LIN {X 0,Y 524.085,Z 47.2,A -85,B 0,C 180,E1 -4854.614,E2 -4854.614} C_VEL
LIN {X 0,Y 524.114,Z 47.199,A -85,B 0,C 180,E1 -4857.694,E2 -4857.694} C_VEL
LIN {X 0,Y 524.126,Z 47.193,A -85,B 0,C 180,E1 -4860.768,E2 -4860.768} C_VEL
LIN {X 0,Y 524.073,Z 47.2,A -85,B 0,C 180,E1 -4863.075,E2 -4863.075} C_VEL
LIN {X 0,Y 524.02,Z 47.208,A -85,B 0,C 180,E1 -4866.159,E2 -4866.159} C_VEL
LIN {X 0,Y 523.989,Z 47.214,A -85,B 0,C 180,E1 -4869.262,E2 -4869.262} C_VEL
LIN {X 0,Y 524.007,Z 47.211,A -85,B 0,C 180,E1 -4871.739,E2 -4871.739} C_VEL
LIN {X 0,Y 523.998,Z 47.213,A -85,B 0,C 180,E1 -4875.052,E2 -4875.052} C_VEL
LIN {X 0,Y 523.949,Z 47.214,A -85,B 0,C 180,E1 -4877.969,E2 -4877.969} C_VEL
LIN {X 0,Y 523.976,Z 47.213,A -85,B 0,C 180,E1 -4880.41,E2 -4880.41} C_VEL
LIN {X 0,Y 523.914,Z 47.225,A -85,B 0,C 180,E1 -4882.893,E2 -4882.893} C_VEL
LIN {X 0,Y 523.938,Z 47.218,A -85,B 0,C 180,E1 -4885.419,E2 -4885.419} C_VEL
LIN {X 0,Y 523.921,Z 47.219,A -85,B 0,C 180,E1 -4888.002,E2 -4888.002} C_VEL
LIN {X 0,Y 523.948,Z 47.22,A -85,B 0,C 180,E1 -4890.854,E2 -4890.854} C_VEL
LIN {X 0,Y 523.932,Z 47.218,A -85,B 0,C 180,E1 -4893.729,E2 -4893.729} C_VEL
LIN {X 0,Y 523.9,Z 47.228,A -85,B 0,C 180,E1 -4896.4,E2 -4896.4} C_VEL
LIN {X 0,Y 523.921,Z 47.219,A -85,B 0,C 180,E1 -4899.085,E2 -4899.085} C_VEL
LIN {X 0,Y 523.942,Z 47.222,A -85,B 0,C 180,E1 -4902.12,E2 -4902.12} C_VEL
LIN {X 0,Y 523.94,Z 47.218,A -85,B 0,C 180,E1 -4905.311,E2 -4905.311} C_VEL
LIN {X 0,Y 523.893,Z 47.223,A -85,B 0,C 180,E1 -4906.9,E2 -4906.9} C_VEL
LIN {X 0,Y 523.23,Z 47.311,A -85,B 0,C 180,E1 -4907.542,E2 -4907.542} C_VEL
LIN {X 0,Y 520.385,Z 47.666,A -85,B 0,C 180,E1 -4908.583,E2 -4908.583} C_VEL
LIN {X 0,Y 517.978,Z 47.966,A -85,B 0,C 180,E1 -4909.423,E2 -4909.423} C_VEL
LIN {X 0,Y 516.946,Z 48.093,A -85,B 0,C 180,E1 -4910.07,E2 -4910.07} C_VEL
LIN {X 0,Y 516.863,Z 48.101,A -85,B 0,C 180,E1 -4910.29,E2 -4910.29} C_VEL
LIN {X 0,Y 516.854,Z 48.105,A -85,B 0,C 180,E1 -4913.347,E2 -4913.347} C_VEL
LIN {X 0,Y 516.885,Z 48.1,A -85,B 0,C 180,E1 -4916.119,E2 -4916.119} C_VEL
LIN {X 0,Y 516.89,Z 48.102,A -85,B 0,C 180,E1 -4918.936,E2 -4918.936} C_VEL
LIN {X 0,Y 516.943,Z 48.197,A -85,B 0,C 180,E1 -4921.475,E2 -4921.475} C_VEL
LIN {X 0,Y 517.512,Z 52.987,A -85,B 0,C 180,E1 -4922.501,E2 -4922.501} C_VEL
LIN {X 0,Y 517.34,Z 63.587,A -85,B 0,C 180,E1 -4924.686,E2 -4924.686} C_VEL
LIN {X 0,Y 519.23,Z 73.369,A -85,B 0,C 180,E1 -4924.897,E2 -4924.897} C_VEL
LIN {X 0,Y 518.679,Z 169.72,A -85,B 0,C 180,E1 -4926.254,E2 -4926.254} C_VEL
LIN {X 0,Y 518.545,Z 182.73,A -85,B 0,C 180,E1 -4926.592,E2 -4926.592} C_VEL
LIN {X 0,Y 518.389,Z 194.491,A -85,B 0,C 180,E1 -4927.042,E2 -4927.042} C_VEL
LIN {X 0,Y 518.056,Z 206.81,A -85,B 0,C 180,E1 -4927.675,E2 -4927.675} C_VEL
LIN {X 0,Y 517.756,Z 217.555,A -85,B 0,C 180,E1 -4928.396,E2 -4928.396} C_VEL
LIN {X 0,Y 517.473,Z 228.558,A -85,B 0,C 180,E1 -4929.322,E2 -4929.322} C_VEL
LIN {X 0,Y 517.175,Z 238.359,A -85,B 0,C 180,E1 -4930.346,E2 -4930.346} C_VEL
LIN {X 0,Y 516.894,Z 247.673,A -85,B 0,C 180,E1 -4931.571,E2 -4931.571} C_VEL
LIN {X 0,Y 516.723,Z 255.105,A -85,B 0,C 180,E1 -4932.793,E2 -4932.793} C_VEL
LIN {X 0,Y 516.573,Z 260.062,A -85,B 0,C 180,E1 -4933.805,E2 -4933.805} C_VEL
LIN {X 0,Y 516.466,Z 264.958,A -85,B 0,C 180,E1 -4935.052,E2 -4935.052} C_VEL
LIN {X 0,Y 516.358,Z 268.425,A -85,B 0,C 180,E1 -4936.22,E2 -4936.22} C_VEL
LIN {X 0,Y 516.301,Z 270.961,A -85,B 0,C 180,E1 -4937.42,E2 -4937.42} C_VEL
LIN {X 0,Y 516.284,Z 272.456,A -85,B 0,C 180,E1 -4938.554,E2 -4938.554} C_VEL
LIN {X 0,Y 516.265,Z 273.148,A -85,B 0,C 180,E1 -4939.807,E2 -4939.807} C_VEL
LIN {X 0,Y 516.232,Z 273.083,A -85,B 0,C 180,E1 -4940.598,E2 -4940.598} C_VEL
LIN {X 0,Y 516.285,Z 272.595,A -85,B 0,C 180,E1 -4941.388,E2 -4941.388} C_VEL
LIN {X 0,Y 516.367,Z 270.394,A -85,B 0,C 180,E1 -4942.964,E2 -4942.964} C_VEL
LIN {X 0,Y 516.433,Z 267.658,A -85,B 0,C 180,E1 -4944.142,E2 -4944.142} C_VEL
LIN {X 0,Y 516.477,Z 263.923,A -85,B 0,C 180,E1 -4945.317,E2 -4945.317} C_VEL
LIN {X 0,Y 516.581,Z 259.084,A -85,B 0,C 180,E1 -4946.49,E2 -4946.49} C_VEL
LIN {X 0,Y 516.689,Z 253.013,A -85,B 0,C 180,E1 -4947.661,E2 -4947.661} C_VEL
LIN {X 0,Y 516.952,Z 245.461,A -85,B 0,C 180,E1 -4948.832,E2 -4948.832} C_VEL
LIN {X 0,Y 517.195,Z 236.016,A -85,B 0,C 180,E1 -4950,E2 -4950} C_VEL
LIN {X 0,Y 517.501,Z 226.287,A -85,B 0,C 180,E1 -4950.973,E2 -4950.973} C_VEL
LIN {X 0,Y 517.809,Z 215.383,A -85,B 0,C 180,E1 -4951.847,E2 -4951.847} C_VEL
LIN {X 0,Y 518.15,Z 204.714,A -85,B 0,C 180,E1 -4952.527,E2 -4952.527} C_VEL
LIN {X 0,Y 518.365,Z 193.027,A -85,B 0,C 180,E1 -4953.109,E2 -4953.109} C_VEL
LIN {X 0,Y 518.526,Z 180.438,A -85,B 0,C 180,E1 -4953.57,E2 -4953.57} C_VEL
LIN {X 0,Y 518.713,Z 168.16,A -85,B 0,C 180,E1 -4953.86,E2 -4953.86} C_VEL
LIN {X 0,Y 519.005,Z 71.995,A -85,B 0,C 180,E1 -4955.214,E2 -4955.214} C_VEL
LIN {X 0,Y 517.288,Z 63.413,A -85,B 0,C 180,E1 -4955.409,E2 -4955.409} C_VEL
LIN {X 0,Y 517.555,Z 52.863,A -85,B 0,C 180,E1 -4957.57,E2 -4957.57} C_VEL
LIN {X 0,Y 516.967,Z 48.094,A -85,B 0,C 180,E1 -4958.6,E2 -4958.6} C_VEL
LIN {X 0,Y 516.954,Z 48.086,A -85,B 0,C 180,E1 -4961.807,E2 -4961.807} C_VEL
LIN {X 0,Y 516.949,Z 48.088,A -85,B 0,C 180,E1 -4965.148,E2 -4965.148} C_VEL
LIN {X 0,Y 516.927,Z 48.095,A -85,B 0,C 180,E1 -4968.222,E2 -4968.222} C_VEL
LIN {X 0,Y 516.914,Z 48.095,A -85,B 0,C 180,E1 -4970.702,E2 -4970.702} C_VEL
LIN {X 0,Y 516.893,Z 48.1,A -85,B 0,C 180,E1 -4974.073,E2 -4974.073} C_VEL
LIN {X 0,Y 516.928,Z 48.091,A -85,B 0,C 180,E1 -4976.658,E2 -4976.658} C_VEL
LIN {X 0,Y 516.913,Z 48.093,A -85,B 0,C 180,E1 -4979.524,E2 -4979.524} C_VEL
LIN {X 0,Y 516.898,Z 48.094,A -85,B 0,C 180,E1 -4982.544,E2 -4982.544} C_VEL
LIN {X 0,Y 516.882,Z 48.097,A -85,B 0,C 180,E1 -4985.332,E2 -4985.332} C_VEL
LIN {X 0,Y 516.883,Z 48.101,A -85,B 0,C 180,E1 -4987.943,E2 -4987.943} C_VEL
LIN {X 0,Y 516.886,Z 48.095,A -85,B 0,C 180,E1 -4990.742,E2 -4990.742} C_VEL
LIN {X 0,Y 516.885,Z 48.095,A -85,B 0,C 180,E1 -4992.832,E2 -4992.832} C_VEL
LIN {X 0,Y 516.898,Z 48.096,A -85,B 0,C 180,E1 -4995.007,E2 -4995.007} C_VEL
LIN {X 0,Y 516.916,Z 48.091,A -85,B 0,C 180,E1 -4998.399,E2 -4998.399} C_VEL
LIN {X 0,Y 516.884,Z 48.103,A -85,B 0,C 180,E1 -5001.284,E2 -5001.284} C_VEL
LIN {X 0,Y 516.876,Z 48.096,A -85,B 0,C 180,E1 -5004.22,E2 -5004.22} C_VEL
LIN {X 0,Y 516.899,Z 48.102,A -85,B 0,C 180,E1 -5007.053,E2 -5007.053} C_VEL
LIN {X 0,Y 516.896,Z 48.093,A -85,B 0,C 180,E1 -5009.797,E2 -5009.797} C_VEL
LIN {X 0,Y 516.931,Z 48.093,A -85,B 0,C 180,E1 -5012.468,E2 -5012.468} C_VEL
LIN {X 0,Y 516.908,Z 48.096,A -85,B 0,C 180,E1 -5015.072,E2 -5015.072} C_VEL
LIN {X 0,Y 516.891,Z 48.1,A -85,B 0,C 180,E1 -5018.463,E2 -5018.463} C_VEL
LIN {X 0,Y 516.899,Z 48.096,A -85,B 0,C 180,E1 -5020.955,E2 -5020.955} C_VEL
LIN {X 0,Y 516.907,Z 48.092,A -85,B 0,C 180,E1 -5023.41,E2 -5023.41} C_VEL
LIN {X 0,Y 516.9,Z 48.095,A -85,B 0,C 180,E1 -5025.834,E2 -5025.834} C_VEL
LIN {X 0,Y 516.972,Z 48.092,A -85,B 0,C 180,E1 -5028.234,E2 -5028.234} C_VEL
LIN {X 0,Y 516.961,Z 48.086,A -85,B 0,C 180,E1 -5031.4,E2 -5031.4} C_VEL
LIN {X 0,Y 517.015,Z 48.083,A -85,B 0,C 180,E1 -5033.757,E2 -5033.757} C_VEL
LIN {X 0,Y 517.086,Z 48.074,A -85,B 0,C 180,E1 -5037.663,E2 -5037.663} C_VEL
LIN {X 0,Y 517.098,Z 48.068,A -85,B 0,C 180,E1 -5040.779,E2 -5040.779} C_VEL
LIN {X 0,Y 517.015,Z 48.08,A -85,B 0,C 180,E1 -5043.117,E2 -5043.117} C_VEL
LIN {X 0,Y 516.982,Z 48.084,A -85,B 0,C 180,E1 -5046.244,E2 -5046.244} C_VEL
LIN {X 0,Y 516.947,Z 48.094,A -85,B 0,C 180,E1 -5049.389,E2 -5049.389} C_VEL
LIN {X 0,Y 516.958,Z 48.089,A -85,B 0,C 180,E1 -5051.807,E2 -5051.807} C_VEL
LIN {X 0,Y 516.951,Z 48.093,A -85,B 0,C 180,E1 -5055.146,E2 -5055.146} C_VEL
LIN {X 0,Y 516.919,Z 48.09,A -85,B 0,C 180,E1 -5058.223,E2 -5058.223} C_VEL
LIN {X 0,Y 516.918,Z 48.094,A -85,B 0,C 180,E1 -5060.701,E2 -5060.701} C_VEL
LIN {X 0,Y 516.895,Z 48.093,A -85,B 0,C 180,E1 -5064.073,E2 -5064.073} C_VEL
LIN {X 0,Y 516.904,Z 48.098,A -85,B 0,C 180,E1 -5066.659,E2 -5066.659} C_VEL
LIN {X 0,Y 516.916,Z 48.091,A -85,B 0,C 180,E1 -5069.524,E2 -5069.524} C_VEL
LIN {X 0,Y 516.899,Z 48.1,A -85,B 0,C 180,E1 -5072.543,E2 -5072.543} C_VEL
LIN {X 0,Y 516.868,Z 48.097,A -85,B 0,C 180,E1 -5075.329,E2 -5075.329} C_VEL
LIN {X 0,Y 516.883,Z 48.097,A -85,B 0,C 180,E1 -5077.943,E2 -5077.943} C_VEL
LIN {X 0,Y 516.887,Z 48.098,A -85,B 0,C 180,E1 -5080.742,E2 -5080.742} C_VEL
LIN {X 0,Y 516.886,Z 48.097,A -85,B 0,C 180,E1 -5082.831,E2 -5082.831} C_VEL
LIN {X 0,Y 516.899,Z 48.093,A -85,B 0,C 180,E1 -5085.007,E2 -5085.007} C_VEL
LIN {X 0,Y 516.913,Z 48.096,A -85,B 0,C 180,E1 -5088.399,E2 -5088.399} C_VEL
LIN {X 0,Y 516.881,Z 48.096,A -85,B 0,C 180,E1 -5091.284,E2 -5091.284} C_VEL
LIN {X 0,Y 516.872,Z 48.101,A -85,B 0,C 180,E1 -5094.219,E2 -5094.219} C_VEL
LIN {X 0,Y 516.885,Z 48.095,A -85,B 0,C 180,E1 -5097.052,E2 -5097.052} C_VEL
LIN {X 0,Y 516.891,Z 48.103,A -85,B 0,C 180,E1 -5099.796,E2 -5099.796} C_VEL
LIN {X 0,Y 516.928,Z 48.092,A -85,B 0,C 180,E1 -5102.467,E2 -5102.467} C_VEL
LIN {X 0,Y 516.956,Z 48.23,A -85,B 0,C 180,E1 -5104.563,E2 -5104.563} C_VEL
LIN {X 0,Y 518.456,Z 56.174,A -85,B 0,C 180,E1 -5105.835,E2 -5105.835} C_VEL
LIN {X 0,Y 518.141,Z 71.265,A -85,B 0,C 180,E1 -5108.099,E2 -5108.099} C_VEL
LIN {X 0,Y 517.746,Z 90.754,A -85,B 0,C 180,E1 -5110.987,E2 -5110.987} C_VEL
LIN {X 0,Y 517.313,Z 110.152,A -85,B 0,C 180,E1 -5113.829,E2 -5113.829} C_VEL
LIN {X 0,Y 517.228,Z 115.912,A -85,B 0,C 180,E1 -5114.631,E2 -5114.631} C_VEL
LIN {X 0,Y 519.045,Z 128.632,A -85,B 0,C 180,E1 -5114.862,E2 -5114.862} C_VEL
LIN {X 0,Y 518.57,Z 224.217,A -85,B 0,C 180,E1 -5116.205,E2 -5116.205} C_VEL
LIN {X 0,Y 518.303,Z 237.571,A -85,B 0,C 180,E1 -5116.548,E2 -5116.548} C_VEL
LIN {X 0,Y 518.026,Z 250.921,A -85,B 0,C 180,E1 -5117.064,E2 -5117.064} C_VEL
LIN {X 0,Y 517.698,Z 262.803,A -85,B 0,C 180,E1 -5117.696,E2 -5117.696} C_VEL
LIN {X 0,Y 517.432,Z 273.773,A -85,B 0,C 180,E1 -5118.443,E2 -5118.443} C_VEL
LIN {X 0,Y 517.159,Z 284.265,A -85,B 0,C 180,E1 -5119.329,E2 -5119.329} C_VEL
LIN {X 0,Y 516.841,Z 292.841,A -85,B 0,C 180,E1 -5120.213,E2 -5120.213} C_VEL
LIN {X 0,Y 516.653,Z 300.762,A -85,B 0,C 180,E1 -5121.197,E2 -5121.197} C_VEL
LIN {X 0,Y 516.502,Z 308.503,A -85,B 0,C 180,E1 -5122.376,E2 -5122.376} C_VEL
LIN {X 0,Y 516.353,Z 315.637,A -85,B 0,C 180,E1 -5123.749,E2 -5123.749} C_VEL
LIN {X 0,Y 516.311,Z 320.386,A -85,B 0,C 180,E1 -5124.924,E2 -5124.924} C_VEL
LIN {X 0,Y 516.369,Z 324.019,A -85,B 0,C 180,E1 -5126.098,E2 -5126.098} C_VEL
LIN {X 0,Y 516.327,Z 325.889,A -85,B 0,C 180,E1 -5126.879,E2 -5126.879} C_VEL
LIN {X 0,Y 516.266,Z 327.289,A -85,B 0,C 180,E1 -5127.659,E2 -5127.659} C_VEL
LIN {X 0,Y 516.189,Z 328.895,A -85,B 0,C 180,E1 -5129.22,E2 -5129.22} C_VEL
LIN {X 0,Y 516.194,Z 329.111,A -85,B 0,C 180,E1 -5130,E2 -5130} C_VEL
LIN {X 0,Y 516.189,Z 328.892,A -85,B 0,C 180,E1 -5130.78,E2 -5130.78} C_VEL
LIN {X 0,Y 516.266,Z 327.279,A -85,B 0,C 180,E1 -5132.341,E2 -5132.341} C_VEL
LIN {X 0,Y 516.327,Z 325.875,A -85,B 0,C 180,E1 -5133.121,E2 -5133.121} C_VEL
LIN {X 0,Y 516.311,Z 322.917,A -85,B 0,C 180,E1 -5134.293,E2 -5134.293} C_VEL
LIN {X 0,Y 516.363,Z 318.916,A -85,B 0,C 180,E1 -5135.467,E2 -5135.467} C_VEL
LIN {X 0,Y 516.406,Z 313.117,A -85,B 0,C 180,E1 -5136.771,E2 -5136.771} C_VEL
LIN {X 0,Y 516.558,Z 306.047,A -85,B 0,C 180,E1 -5138.016,E2 -5138.016} C_VEL
LIN {X 0,Y 516.724,Z 297.714,A -85,B 0,C 180,E1 -5139.196,E2 -5139.196} C_VEL
LIN {X 0,Y 516.941,Z 289.178,A -85,B 0,C 180,E1 -5140.18,E2 -5140.18} C_VEL
LIN {X 0,Y 517.291,Z 278.64,A -85,B 0,C 180,E1 -5141.163,E2 -5141.163} C_VEL
LIN {X 0,Y 517.566,Z 267.025,A -85,B 0,C 180,E1 -5142.034,E2 -5142.034} C_VEL
LIN {X 0,Y 517.903,Z 254.859,A -85,B 0,C 180,E1 -5142.739,E2 -5142.739} C_VEL
LIN {X 0,Y 518.195,Z 242.464,A -85,B 0,C 180,E1 -5143.28,E2 -5143.28} C_VEL
LIN {X 0,Y 518.456,Z 229.739,A -85,B 0,C 180,E1 -5143.673,E2 -5143.673} C_VEL
LIN {X 0,Y 518.648,Z 214.605,A -85,B 0,C 180,E1 -5143.942,E2 -5143.942} C_VEL
LIN {X 0,Y 518.957,Z 128.068,A -85,B 0,C 180,E1 -5145.147,E2 -5145.147} C_VEL
LIN {X 0,Y 517.216,Z 115.441,A -85,B 0,C 180,E1 -5145.386,E2 -5145.386} C_VEL
LIN {X 0,Y 517.714,Z 93.474,A -85,B 0,C 180,E1 -5148.603,E2 -5148.603} C_VEL
LIN {X 0,Y 518.102,Z 74.124,A -85,B 0,C 180,E1 -5151.485,E2 -5151.485} C_VEL
LIN {X 0,Y 518.546,Z 56.468,A -85,B 0,C 180,E1 -5154.16,E2 -5154.16} C_VEL
LIN {X 0,Y 516.956,Z 48.092,A -85,B 0,C 180,E1 -5155.572,E2 -5155.572} C_VEL
LIN {X 0,Y 516.919,Z 48.098,A -85,B 0,C 180,E1 -5158.415,E2 -5158.415} C_VEL
LIN {X 0,Y 516.892,Z 48.095,A -85,B 0,C 180,E1 -5161.11,E2 -5161.11} C_VEL
LIN {X 0,Y 516.89,Z 48.102,A -85,B 0,C 180,E1 -5163.963,E2 -5163.963} C_VEL
LIN {X 0,Y 516.88,Z 48.097,A -85,B 0,C 180,E1 -5166.746,E2 -5166.746} C_VEL
LIN {X 0,Y 516.885,Z 48.098,A -85,B 0,C 180,E1 -5169.721,E2 -5169.721} C_VEL
LIN {X 0,Y 516.915,Z 48.099,A -85,B 0,C 180,E1 -5171.775,E2 -5171.775} C_VEL
LIN {X 0,Y 516.898,Z 48.093,A -85,B 0,C 180,E1 -5175.007,E2 -5175.007} C_VEL
LIN {X 0,Y 516.917,Z 48.09,A -85,B 0,C 180,E1 -5178.399,E2 -5178.399} C_VEL
LIN {X 0,Y 516.884,Z 48.1,A -85,B 0,C 180,E1 -5181.284,E2 -5181.284} C_VEL
LIN {X 0,Y 516.875,Z 48.096,A -85,B 0,C 180,E1 -5184.22,E2 -5184.22} C_VEL
LIN {X 0,Y 516.885,Z 48.1,A -85,B 0,C 180,E1 -5187.052,E2 -5187.052} C_VEL
LIN {X 0,Y 516.896,Z 48.092,A -85,B 0,C 180,E1 -5189.796,E2 -5189.796} C_VEL
LIN {X 0,Y 516.931,Z 48.092,A -85,B 0,C 180,E1 -5192.467,E2 -5192.467} C_VEL
LIN {X 0,Y 516.908,Z 48.098,A -85,B 0,C 180,E1 -5195.072,E2 -5195.072} C_VEL
LIN {X 0,Y 516.89,Z 48.098,A -85,B 0,C 180,E1 -5198.462,E2 -5198.462} C_VEL
LIN {X 0,Y 516.899,Z 48.097,A -85,B 0,C 180,E1 -5200.955,E2 -5200.955} C_VEL
LIN {X 0,Y 516.915,Z 48.089,A -85,B 0,C 180,E1 -5203.41,E2 -5203.41} C_VEL
LIN {X 0,Y 516.899,Z 48.095,A -85,B 0,C 180,E1 -5205.834,E2 -5205.834} C_VEL
LIN {X 0,Y 516.971,Z 48.089,A -85,B 0,C 180,E1 -5208.234,E2 -5208.234} C_VEL
LIN {X 0,Y 516.97,Z 48.085,A -85,B 0,C 180,E1 -5211.4,E2 -5211.4} C_VEL
LIN {X 0,Y 517.014,Z 48.079,A -85,B 0,C 180,E1 -5213.757,E2 -5213.757} C_VEL
LIN {X 0,Y 517.085,Z 48.074,A -85,B 0,C 180,E1 -5217.663,E2 -5217.663} C_VEL
LIN {X 0,Y 517.097,Z 48.069,A -85,B 0,C 180,E1 -5220.779,E2 -5220.779} C_VEL
LIN {X 0,Y 517.014,Z 48.079,A -85,B 0,C 180,E1 -5223.117,E2 -5223.117} C_VEL
LIN {X 0,Y 516.989,Z 48.083,A -85,B 0,C 180,E1 -5226.243,E2 -5226.243} C_VEL
LIN {X 0,Y 516.945,Z 48.092,A -85,B 0,C 180,E1 -5229.389,E2 -5229.389} C_VEL
LIN {X 0,Y 516.957,Z 48.089,A -85,B 0,C 180,E1 -5231.807,E2 -5231.807} C_VEL
LIN {X 0,Y 516.949,Z 48.092,A -85,B 0,C 180,E1 -5235.146,E2 -5235.146} C_VEL
LIN {X 0,Y 516.917,Z 48.09,A -85,B 0,C 180,E1 -5238.222,E2 -5238.222} C_VEL
LIN {X 0,Y 516.916,Z 48.096,A -85,B 0,C 180,E1 -5240.701,E2 -5240.701} C_VEL
LIN {X 0,Y 516.906,Z 48.092,A -85,B 0,C 180,E1 -5244.072,E2 -5244.072} C_VEL
LIN {X 0,Y 516.901,Z 48.1,A -85,B 0,C 180,E1 -5246.659,E2 -5246.659} C_VEL
LIN {X 0,Y 516.913,Z 48.092,A -85,B 0,C 180,E1 -5249.523,E2 -5249.523} C_VEL
LIN {X 0,Y 516.897,Z 48.101,A -85,B 0,C 180,E1 -5252.543,E2 -5252.543} C_VEL
LIN {X 0,Y 516.864,Z 48.098,A -85,B 0,C 180,E1 -5255.329,E2 -5255.329} C_VEL
LIN {X 0,Y 516.881,Z 48.099,A -85,B 0,C 180,E1 -5257.943,E2 -5257.943} C_VEL
LIN {X 0,Y 516.873,Z 48.094,A -85,B 0,C 180,E1 -5260.743,E2 -5260.743} C_VEL
LIN {X 0,Y 516.883,Z 48.103,A -85,B 0,C 180,E1 -5263.893,E2 -5263.893} C_VEL
LIN {X 0,Y 516.846,Z 48.101,A -85,B 0,C 180,E1 -5266.901,E2 -5266.901} C_VEL
LIN {X 0,Y 516.886,Z 48.102,A -85,B 0,C 180,E1 -5269.59,E2 -5269.59} C_VEL
LIN {X 0,Y 516.863,Z 48.101,A -85,B 0,C 180,E1 -5270.29,E2 -5270.29} C_VEL
LIN {X 0,Y 516.199,Z 48.182,A -85,B 0,C 180,E1 -5270.94,E2 -5270.94} C_VEL
LIN {X 0,Y 513.349,Z 48.543,A -85,B 0,C 180,E1 -5271.996,E2 -5271.996} C_VEL
LIN {X 0,Y 510.936,Z 48.848,A -85,B 0,C 180,E1 -5272.846,E2 -5272.846} C_VEL
LIN {X 0,Y 509.894,Z 48.976,A -85,B 0,C 180,E1 -5273.503,E2 -5273.503} C_VEL
LIN {X 0,Y 509.807,Z 48.984,A -85,B 0,C 180,E1 -5273.725,E2 -5273.725} C_VEL
LIN {X 0,Y 509.843,Z 48.976,A -85,B 0,C 180,E1 -5276.538,E2 -5276.538} C_VEL
LIN {X 0,Y 509.841,Z 48.982,A -85,B 0,C 180,E1 -5279.334,E2 -5279.334} C_VEL
LIN {X 0,Y 509.924,Z 49.163,A -85,B 0,C 180,E1 -5281.344,E2 -5281.344} C_VEL
LIN {X 0,Y 510.522,Z 54.689,A -85,B 0,C 180,E1 -5282.537,E2 -5282.537} C_VEL
LIN {X 0,Y 510.374,Z 63.959,A -85,B 0,C 180,E1 -5284.464,E2 -5284.464} C_VEL
LIN {X 0,Y 512.396,Z 74.105,A -85,B 0,C 180,E1 -5284.688,E2 -5284.688} C_VEL
LIN {X 0,Y 511.831,Z 169.609,A -85,B 0,C 180,E1 -5286.051,E2 -5286.051} C_VEL
LIN {X 0,Y 511.668,Z 182.796,A -85,B 0,C 180,E1 -5286.392,E2 -5286.392} C_VEL
LIN {X 0,Y 511.491,Z 194.615,A -85,B 0,C 180,E1 -5286.848,E2 -5286.848} C_VEL
LIN {X 0,Y 511.164,Z 206.558,A -85,B 0,C 180,E1 -5287.465,E2 -5287.465} C_VEL
LIN {X 0,Y 510.842,Z 217.454,A -85,B 0,C 180,E1 -5288.194,E2 -5288.194} C_VEL
LIN {X 0,Y 510.543,Z 227.421,A -85,B 0,C 180,E1 -5289.028,E2 -5289.028} C_VEL
LIN {X 0,Y 510.239,Z 237.494,A -85,B 0,C 180,E1 -5290.068,E2 -5290.068} C_VEL
LIN {X 0,Y 509.956,Z 245.666,A -85,B 0,C 180,E1 -5291.103,E2 -5291.103} C_VEL
LIN {X 0,Y 509.706,Z 253.551,A -85,B 0,C 180,E1 -5292.341,E2 -5292.341} C_VEL
LIN {X 0,Y 509.531,Z 259.805,A -85,B 0,C 180,E1 -5293.575,E2 -5293.575} C_VEL
LIN {X 0,Y 509.384,Z 265.306,A -85,B 0,C 180,E1 -5294.971,E2 -5294.971} C_VEL
LIN {X 0,Y 509.321,Z 268.434,A -85,B 0,C 180,E1 -5296.026,E2 -5296.026} C_VEL
LIN {X 0,Y 509.214,Z 271.091,A -85,B 0,C 180,E1 -5297.242,E2 -5297.242} C_VEL
LIN {X 0,Y 509.211,Z 272.807,A -85,B 0,C 180,E1 -5298.5,E2 -5298.5} C_VEL
LIN {X 0,Y 509.197,Z 273.504,A -85,B 0,C 180,E1 -5299.664,E2 -5299.664} C_VEL
LIN {X 0,Y 509.183,Z 273.096,A -85,B 0,C 180,E1 -5301.267,E2 -5301.267} C_VEL
LIN {X 0,Y 509.231,Z 272.268,A -85,B 0,C 180,E1 -5302.067,E2 -5302.067} C_VEL
LIN {X 0,Y 509.318,Z 269.817,A -85,B 0,C 180,E1 -5303.473,E2 -5303.473} C_VEL
LIN {X 0,Y 509.327,Z 266.123,A -85,B 0,C 180,E1 -5304.854,E2 -5304.854} C_VEL
LIN {X 0,Y 509.501,Z 261.783,A -85,B 0,C 180,E1 -5306.045,E2 -5306.045} C_VEL
LIN {X 0,Y 509.555,Z 256.296,A -85,B 0,C 180,E1 -5307.233,E2 -5307.233} C_VEL
LIN {X 0,Y 509.829,Z 249.438,A -85,B 0,C 180,E1 -5308.42,E2 -5308.42} C_VEL
LIN {X 0,Y 510.083,Z 240.879,A -85,B 0,C 180,E1 -5309.605,E2 -5309.605} C_VEL
LIN {X 0,Y 510.324,Z 232.146,A -85,B 0,C 180,E1 -5310.592,E2 -5310.592} C_VEL
LIN {X 0,Y 510.708,Z 221.386,A -85,B 0,C 180,E1 -5311.577,E2 -5311.577} C_VEL
LIN {X 0,Y 511.043,Z 210.526,A -85,B 0,C 180,E1 -5312.365,E2 -5312.365} C_VEL
LIN {X 0,Y 511.349,Z 198.405,A -85,B 0,C 180,E1 -5313.053,E2 -5313.053} C_VEL
LIN {X 0,Y 511.588,Z 185.604,A -85,B 0,C 180,E1 -5313.594,E2 -5313.594} C_VEL
LIN {X 0,Y 511.751,Z 172.634,A -85,B 0,C 180,E1 -5313.962,E2 -5313.962} C_VEL
LIN {X 0,Y 511.935,Z 152.544,A -85,B 0,C 180,E1 -5314.281,E2 -5314.281} C_VEL
LIN {X 0,Y 512.204,Z 73.139,A -85,B 0,C 180,E1 -5315.404,E2 -5315.404} C_VEL
LIN {X 0,Y 510.315,Z 63.795,A -85,B 0,C 180,E1 -5315.607,E2 -5315.607} C_VEL
LIN {X 0,Y 510.561,Z 53.878,A -85,B 0,C 180,E1 -5317.651,E2 -5317.651} C_VEL
LIN {X 0,Y 509.913,Z 48.973,A -85,B 0,C 180,E1 -5318.72,E2 -5318.72} C_VEL
LIN {X 0,Y 509.906,Z 48.964,A -85,B 0,C 180,E1 -5321.932,E2 -5321.932} C_VEL
LIN {X 0,Y 509.896,Z 48.966,A -85,B 0,C 180,E1 -5325.242,E2 -5325.242} C_VEL
LIN {X 0,Y 509.884,Z 48.97,A -85,B 0,C 180,E1 -5327.999,E2 -5327.999} C_VEL
LIN {X 0,Y 509.852,Z 48.972,A -85,B 0,C 180,E1 -5331.002,E2 -5331.002} C_VEL
LIN {X 0,Y 509.824,Z 48.975,A -85,B 0,C 180,E1 -5333.564,E2 -5333.564} C_VEL
LIN {X 0,Y 509.914,Z 48.968,A -85,B 0,C 180,E1 -5336.379,E2 -5336.379} C_VEL
LIN {X 0,Y 509.879,Z 48.968,A -85,B 0,C 180,E1 -5338.844,E2 -5338.844} C_VEL
LIN {X 0,Y 509.823,Z 48.978,A -85,B 0,C 180,E1 -5341.59,E2 -5341.59} C_VEL
LIN {X 0,Y 509.855,Z 48.972,A -85,B 0,C 180,E1 -5344.414,E2 -5344.414} C_VEL
LIN {X 0,Y 509.821,Z 48.978,A -85,B 0,C 180,E1 -5347.341,E2 -5347.341} C_VEL
LIN {X 0,Y 509.841,Z 48.973,A -85,B 0,C 180,E1 -5350.382,E2 -5350.382} C_VEL
LIN {X 0,Y 509.825,Z 48.977,A -85,B 0,C 180,E1 -5353.062,E2 -5353.062} C_VEL
LIN {X 0,Y 509.825,Z 48.978,A -85,B 0,C 180,E1 -5355.794,E2 -5355.794} C_VEL
LIN {X 0,Y 509.858,Z 48.971,A -85,B 0,C 180,E1 -5358.575,E2 -5358.575} C_VEL
LIN {X 0,Y 509.854,Z 48.972,A -85,B 0,C 180,E1 -5361.787,E2 -5361.787} C_VEL
LIN {X 0,Y 509.836,Z 48.975,A -85,B 0,C 180,E1 -5364.622,E2 -5364.622} C_VEL
LIN {X 0,Y 509.865,Z 48.972,A -85,B 0,C 180,E1 -5367.481,E2 -5367.481} C_VEL
LIN {X 0,Y 509.863,Z 48.971,A -85,B 0,C 180,E1 -5370.274,E2 -5370.274} C_VEL
LIN {X 0,Y 509.888,Z 48.973,A -85,B 0,C 180,E1 -5372.945,E2 -5372.945} C_VEL
LIN {X 0,Y 509.86,Z 48.97,A -85,B 0,C 180,E1 -5375.574,E2 -5375.574} C_VEL
LIN {X 0,Y 509.855,Z 48.974,A -85,B 0,C 180,E1 -5378.999,E2 -5378.999} C_VEL
LIN {X 0,Y 509.863,Z 48.969,A -85,B 0,C 180,E1 -5381.516,E2 -5381.516} C_VEL
LIN {X 0,Y 509.916,Z 48.966,A -85,B 0,C 180,E1 -5384.819,E2 -5384.819} C_VEL
LIN {X 0,Y 509.907,Z 48.97,A -85,B 0,C 180,E1 -5388.124,E2 -5388.124} C_VEL
LIN {X 0,Y 509.909,Z 48.964,A -85,B 0,C 180,E1 -5391.28,E2 -5391.28} C_VEL
LIN {X 0,Y 509.965,Z 48.96,A -85,B 0,C 180,E1 -5393.67,E2 -5393.67} C_VEL
LIN {X 0,Y 510.056,Z 48.95,A -85,B 0,C 180,E1 -5397.631,E2 -5397.631} C_VEL
LIN {X 0,Y 510.061,Z 48.951,A -85,B 0,C 180,E1 -5400,E2 -5400} C_VEL
LIN {X 0,Y 510.058,Z 48.947,A -85,B 0,C 180,E1 -5402.369,E2 -5402.369} C_VEL
LIN {X 0,Y 509.972,Z 48.963,A -85,B 0,C 180,E1 -5405.536,E2 -5405.536} C_VEL
LIN {X 0,Y 509.909,Z 48.964,A -85,B 0,C 180,E1 -5408.72,E2 -5408.72} C_VEL
LIN {X 0,Y 509.91,Z 48.966,A -85,B 0,C 180,E1 -5411.932,E2 -5411.932} C_VEL
LIN {X 0,Y 509.9,Z 48.973,A -85,B 0,C 180,E1 -5415.242,E2 -5415.242} C_VEL
LIN {X 0,Y 509.864,Z 48.97,A -85,B 0,C 180,E1 -5418.484,E2 -5418.484} C_VEL
LIN {X 0,Y 509.856,Z 48.978,A -85,B 0,C 180,E1 -5421.002,E2 -5421.002} C_VEL
LIN {X 0,Y 509.827,Z 48.976,A -85,B 0,C 180,E1 -5423.564,E2 -5423.564} C_VEL
LIN {X 0,Y 509.89,Z 48.968,A -85,B 0,C 180,E1 -5426.372,E2 -5426.372} C_VEL
LIN {X 0,Y 509.864,Z 48.969,A -85,B 0,C 180,E1 -5429.726,E2 -5429.726} C_VEL
LIN {X 0,Y 509.871,Z 48.976,A -85,B 0,C 180,E1 -5432.773,E2 -5432.773} C_VEL
LIN {X 0,Y 509.827,Z 48.974,A -85,B 0,C 180,E1 -5435.578,E2 -5435.578} C_VEL
LIN {X 0,Y 509.853,Z 48.977,A -85,B 0,C 180,E1 -5438.338,E2 -5438.338} C_VEL
LIN {X 0,Y 509.859,Z 48.97,A -85,B 0,C 180,E1 -5441.425,E2 -5441.425} C_VEL
LIN {X 0,Y 509.843,Z 48.975,A -85,B 0,C 180,E1 -5444.67,E2 -5444.67} C_VEL
LIN {X 0,Y 509.853,Z 48.979,A -85,B 0,C 180,E1 -5448.104,E2 -5448.104} C_VEL
LIN {X 0,Y 509.842,Z 48.973,A -85,B 0,C 180,E1 -5450.647,E2 -5450.647} C_VEL
LIN {X 0,Y 509.813,Z 48.98,A -85,B 0,C 180,E1 -5453.645,E2 -5453.645} C_VEL
LIN {X 0,Y 509.846,Z 48.972,A -85,B 0,C 180,E1 -5456.538,E2 -5456.538} C_VEL
LIN {X 0,Y 509.846,Z 48.975,A -85,B 0,C 180,E1 -5459.334,E2 -5459.334} C_VEL
LIN {X 0,Y 509.893,Z 48.971,A -85,B 0,C 180,E1 -5462.054,E2 -5462.054} C_VEL
LIN {X 0,Y 509.952,Z 49.138,A -85,B 0,C 180,E1 -5464.407,E2 -5464.407} C_VEL
LIN {X 0,Y 511.537,Z 58.216,A -85,B 0,C 180,E1 -5465.874,E2 -5465.874} C_VEL
LIN {X 0,Y 511.088,Z 76.393,A -85,B 0,C 180,E1 -5468.629,E2 -5468.629} C_VEL
LIN {X 0,Y 510.608,Z 98.096,A -85,B 0,C 180,E1 -5471.875,E2 -5471.875} C_VEL
LIN {X 0,Y 510.177,Z 115.209,A -85,B 0,C 180,E1 -5474.408,E2 -5474.408} C_VEL
LIN {X 0,Y 512.138,Z 129.834,A -85,B 0,C 180,E1 -5474.679,E2 -5474.679} C_VEL
LIN {X 0,Y 511.691,Z 223.748,A -85,B 0,C 180,E1 -5476.016,E2 -5476.016} C_VEL
LIN {X 0,Y 511.424,Z 236.376,A -85,B 0,C 180,E1 -5476.338,E2 -5476.338} C_VEL
LIN {X 0,Y 511.103,Z 249.378,A -85,B 0,C 180,E1 -5476.835,E2 -5476.835} C_VEL
LIN {X 0,Y 510.791,Z 261.177,A -85,B 0,C 180,E1 -5477.45,E2 -5477.45} C_VEL
LIN {X 0,Y 510.419,Z 272.08,A -85,B 0,C 180,E1 -5478.181,E2 -5478.181} C_VEL
LIN {X 0,Y 510.126,Z 282.798,A -85,B 0,C 180,E1 -5479.08,E2 -5479.08} C_VEL
LIN {X 0,Y 509.804,Z 292.454,A -85,B 0,C 180,E1 -5480.077,E2 -5480.077} C_VEL
LIN {X 0,Y 509.601,Z 300.377,A -85,B 0,C 180,E1 -5481.074,E2 -5481.074} C_VEL
LIN {X 0,Y 509.415,Z 308.117,A -85,B 0,C 180,E1 -5482.269,E2 -5482.269} C_VEL
LIN {X 0,Y 509.26,Z 315.252,A -85,B 0,C 180,E1 -5483.661,E2 -5483.661} C_VEL
LIN {X 0,Y 509.239,Z 320.003,A -85,B 0,C 180,E1 -5484.853,E2 -5484.853} C_VEL
LIN {X 0,Y 509.275,Z 323.635,A -85,B 0,C 180,E1 -5486.043,E2 -5486.043} C_VEL
LIN {X 0,Y 509.241,Z 325.506,A -85,B 0,C 180,E1 -5486.835,E2 -5486.835} C_VEL
LIN {X 0,Y 509.196,Z 326.907,A -85,B 0,C 180,E1 -5487.627,E2 -5487.627} C_VEL
LIN {X 0,Y 509.101,Z 328.512,A -85,B 0,C 180,E1 -5489.209,E2 -5489.209} C_VEL
LIN {X 0,Y 509.105,Z 328.727,A -85,B 0,C 180,E1 -5490,E2 -5490} C_VEL
LIN {X 0,Y 509.12,Z 327.895,A -85,B 0,C 180,E1 -5491.582,E2 -5491.582} C_VEL
LIN {X 0,Y 509.196,Z 326.894,A -85,B 0,C 180,E1 -5492.373,E2 -5492.373} C_VEL
LIN {X 0,Y 509.241,Z 325.488,A -85,B 0,C 180,E1 -5493.165,E2 -5493.165} C_VEL
LIN {X 0,Y 509.204,Z 322.527,A -85,B 0,C 180,E1 -5494.354,E2 -5494.354} C_VEL
LIN {X 0,Y 509.273,Z 318.526,A -85,B 0,C 180,E1 -5495.543,E2 -5495.543} C_VEL
LIN {X 0,Y 509.33,Z 312.473,A -85,B 0,C 180,E1 -5496.915,E2 -5496.915} C_VEL
LIN {X 0,Y 509.477,Z 305.652,A -85,B 0,C 180,E1 -5498.129,E2 -5498.129} C_VEL
LIN {X 0,Y 509.681,Z 297.318,A -85,B 0,C 180,E1 -5499.324,E2 -5499.324} C_VEL
LIN {X 0,Y 509.926,Z 288.78,A -85,B 0,C 180,E1 -5500.321,E2 -5500.321} C_VEL
LIN {X 0,Y 510.288,Z 278.245,A -85,B 0,C 180,E1 -5501.318,E2 -5501.318} C_VEL
LIN {X 0,Y 510.566,Z 267.39,A -85,B 0,C 180,E1 -5502.148,E2 -5502.148} C_VEL
LIN {X 0,Y 510.917,Z 256.416,A -85,B 0,C 180,E1 -5502.815,E2 -5502.815} C_VEL
LIN {X 0,Y 511.203,Z 244.706,A -85,B 0,C 180,E1 -5503.364,E2 -5503.364} C_VEL
LIN {X 0,Y 511.536,Z 231.231,A -85,B 0,C 180,E1 -5503.811,E2 -5503.811} C_VEL
LIN {X 0,Y 511.778,Z 217.909,A -85,B 0,C 180,E1 -5504.083,E2 -5504.083} C_VEL
LIN {X 0,Y 512.001,Z 128.019,A -85,B 0,C 180,E1 -5505.357,E2 -5505.357} C_VEL
LIN {X 0,Y 510.189,Z 115.04,A -85,B 0,C 180,E1 -5505.609,E2 -5505.609} C_VEL
LIN {X 0,Y 510.715,Z 93.16,A -85,B 0,C 180,E1 -5508.868,E2 -5508.868} C_VEL
LIN {X 0,Y 511.169,Z 75.235,A -85,B 0,C 180,E1 -5511.579,E2 -5511.579} C_VEL
LIN {X 0,Y 511.67,Z 58.709,A -85,B 0,C 180,E1 -5514.119,E2 -5514.119} C_VEL
LIN {X 0,Y 509.913,Z 48.971,A -85,B 0,C 180,E1 -5515.759,E2 -5515.759} C_VEL
LIN {X 0,Y 509.878,Z 48.971,A -85,B 0,C 180,E1 -5518.844,E2 -5518.844} C_VEL
LIN {X 0,Y 509.823,Z 48.976,A -85,B 0,C 180,E1 -5521.59,E2 -5521.59} C_VEL
LIN {X 0,Y 509.842,Z 48.978,A -85,B 0,C 180,E1 -5524.414,E2 -5524.414} C_VEL
LIN {X 0,Y 509.82,Z 48.977,A -85,B 0,C 180,E1 -5527.341,E2 -5527.341} C_VEL
LIN {X 0,Y 509.841,Z 48.975,A -85,B 0,C 180,E1 -5530.382,E2 -5530.382} C_VEL
LIN {X 0,Y 509.827,Z 48.974,A -85,B 0,C 180,E1 -5533.062,E2 -5533.062} C_VEL
LIN {X 0,Y 509.826,Z 48.979,A -85,B 0,C 180,E1 -5535.793,E2 -5535.793} C_VEL
LIN {X 0,Y 509.859,Z 48.969,A -85,B 0,C 180,E1 -5538.575,E2 -5538.575} C_VEL
LIN {X 0,Y 509.854,Z 48.973,A -85,B 0,C 180,E1 -5541.787,E2 -5541.787} C_VEL
LIN {X 0,Y 509.833,Z 48.974,A -85,B 0,C 180,E1 -5544.622,E2 -5544.622} C_VEL
LIN {X 0,Y 509.864,Z 48.974,A -85,B 0,C 180,E1 -5547.481,E2 -5547.481} C_VEL
LIN {X 0,Y 509.863,Z 48.968,A -85,B 0,C 180,E1 -5550.274,E2 -5550.274} C_VEL
LIN {X 0,Y 509.888,Z 48.973,A -85,B 0,C 180,E1 -5552.944,E2 -5552.944} C_VEL
LIN {X 0,Y 509.859,Z 48.971,A -85,B 0,C 180,E1 -5555.573,E2 -5555.573} C_VEL
LIN {X 0,Y 509.855,Z 48.974,A -85,B 0,C 180,E1 -5558.998,E2 -5558.998} C_VEL
LIN {X 0,Y 509.885,Z 48.968,A -85,B 0,C 180,E1 -5562.002,E2 -5562.002} C_VEL
LIN {X 0,Y 509.916,Z 48.967,A -85,B 0,C 180,E1 -5564.819,E2 -5564.819} C_VEL
LIN {X 0,Y 509.906,Z 48.968,A -85,B 0,C 180,E1 -5568.124,E2 -5568.124} C_VEL
LIN {X 0,Y 509.916,Z 48.963,A -85,B 0,C 180,E1 -5571.28,E2 -5571.28} C_VEL
LIN {X 0,Y 509.964,Z 48.956,A -85,B 0,C 180,E1 -5573.67,E2 -5573.67} C_VEL
LIN {X 0,Y 510.055,Z 48.95,A -85,B 0,C 180,E1 -5577.631,E2 -5577.631} C_VEL
LIN {X 0,Y 510.06,Z 48.952,A -85,B 0,C 180,E1 -5580,E2 -5580} C_VEL
LIN {X 0,Y 510.057,Z 48.945,A -85,B 0,C 180,E1 -5582.369,E2 -5582.369} C_VEL
LIN {X 0,Y 509.972,Z 48.963,A -85,B 0,C 180,E1 -5585.536,E2 -5585.536} C_VEL
LIN {X 0,Y 509.925,Z 48.962,A -85,B 0,C 180,E1 -5587.922,E2 -5587.922} C_VEL
LIN {X 0,Y 509.917,Z 48.968,A -85,B 0,C 180,E1 -5591.125,E2 -5591.125} C_VEL
LIN {X 0,Y 509.867,Z 48.967,A -85,B 0,C 180,E1 -5594.366,E2 -5594.366} C_VEL
LIN {X 0,Y 509.875,Z 48.973,A -85,B 0,C 180,E1 -5596.826,E2 -5596.826} C_VEL
LIN {X 0,Y 509.92,Z 48.963,A -85,B 0,C 180,E1 -5600.155,E2 -5600.155} C_VEL
LIN {X 0,Y 509.833,Z 48.973,A -85,B 0,C 180,E1 -5603.563,E2 -5603.563} C_VEL
LIN {X 0,Y 509.882,Z 48.971,A -85,B 0,C 180,E1 -5606.371,E2 -5606.371} C_VEL
LIN {X 0,Y 509.862,Z 48.97,A -85,B 0,C 180,E1 -5609.726,E2 -5609.726} C_VEL
LIN {X 0,Y 509.87,Z 48.973,A -85,B 0,C 180,E1 -5612.773,E2 -5612.773} C_VEL
LIN {X 0,Y 509.824,Z 48.976,A -85,B 0,C 180,E1 -5615.578,E2 -5615.578} C_VEL
LIN {X 0,Y 509.851,Z 48.979,A -85,B 0,C 180,E1 -5618.338,E2 -5618.338} C_VEL
LIN {X 0,Y 509.847,Z 48.968,A -85,B 0,C 180,E1 -5621.426,E2 -5621.426} C_VEL
LIN {X 0,Y 509.841,Z 48.975,A -85,B 0,C 180,E1 -5624.67,E2 -5624.67} C_VEL
LIN {X 0,Y 509.85,Z 48.978,A -85,B 0,C 180,E1 -5628.104,E2 -5628.104} C_VEL
LIN {X 0,Y 509.835,Z 48.974,A -85,B 0,C 180,E1 -5630.646,E2 -5630.646} C_VEL
LIN {X 0,Y 509.807,Z 48.984,A -85,B 0,C 180,E1 -5633.725,E2 -5633.725} C_VEL
LIN {X 0,Y 509.147,Z 49.063,A -85,B 0,C 180,E1 -5634.385,E2 -5634.385} C_VEL
LIN {X 0,Y 506.341,Z 49.417,A -85,B 0,C 180,E1 -5635.457,E2 -5635.457} C_VEL
LIN {X 0,Y 503.954,Z 49.714,A -85,B 0,C 180,E1 -5636.321,E2 -5636.321} C_VEL
LIN {X 0,Y 502.906,Z 49.843,A -85,B 0,C 180,E1 -5636.987,E2 -5636.987} C_VEL
LIN {X 0,Y 502.808,Z 49.854,A -85,B 0,C 180,E1 -5637.213,E2 -5637.213} C_VEL
LIN {X 0,Y 502.815,Z 49.855,A -85,B 0,C 180,E1 -5640.065,E2 -5640.065} C_VEL
LIN {X 0,Y 502.876,Z 50.003,A -85,B 0,C 180,E1 -5641.174,E2 -5641.174} C_VEL
LIN {X 0,Y 503.575,Z 55.366,A -85,B 0,C 180,E1 -5642.351,E2 -5642.351} C_VEL
LIN {X 0,Y 503.472,Z 64.587,A -85,B 0,C 180,E1 -5644.245,E2 -5644.245} C_VEL
LIN {X 0,Y 505.584,Z 75.16,A -85,B 0,C 180,E1 -5644.474,E2 -5644.474} C_VEL
LIN {X 0,Y 504.991,Z 169.7,A -85,B 0,C 180,E1 -5645.842,E2 -5645.842} C_VEL
LIN {X 0,Y 504.828,Z 183.02,A -85,B 0,C 180,E1 -5646.189,E2 -5646.189} C_VEL
LIN {X 0,Y 504.624,Z 195.439,A -85,B 0,C 180,E1 -5646.676,E2 -5646.676} C_VEL
LIN {X 0,Y 504.303,Z 206.376,A -85,B 0,C 180,E1 -5647.249,E2 -5647.249} C_VEL
LIN {X 0,Y 503.94,Z 217.411,A -85,B 0,C 180,E1 -5647.988,E2 -5647.988} C_VEL
LIN {X 0,Y 503.594,Z 228.076,A -85,B 0,C 180,E1 -5648.893,E2 -5648.893} C_VEL
LIN {X 0,Y 503.255,Z 238.491,A -85,B 0,C 180,E1 -5649.992,E2 -5649.992} C_VEL
LIN {X 0,Y 502.945,Z 246.541,A -85,B 0,C 180,E1 -5651.041,E2 -5651.041} C_VEL
LIN {X 0,Y 502.68,Z 254.309,A -85,B 0,C 180,E1 -5652.297,E2 -5652.297} C_VEL
LIN {X 0,Y 502.446,Z 261.407,A -85,B 0,C 180,E1 -5653.755,E2 -5653.755} C_VEL
LIN {X 0,Y 502.331,Z 265.621,A -85,B 0,C 180,E1 -5654.876,E2 -5654.876} C_VEL
LIN {X 0,Y 502.196,Z 269.513,A -85,B 0,C 180,E1 -5656.237,E2 -5656.237} C_VEL
LIN {X 0,Y 502.154,Z 271.224,A -85,B 0,C 180,E1 -5657.06,E2 -5657.06} C_VEL
LIN {X 0,Y 502.125,Z 273.167,A -85,B 0,C 180,E1 -5658.452,E2 -5658.452} C_VEL
LIN {X 0,Y 502.12,Z 273.861,A -85,B 0,C 180,E1 -5659.516,E2 -5659.516} C_VEL
LIN {X 0,Y 502.096,Z 273.563,A -85,B 0,C 180,E1 -5661.143,E2 -5661.143} C_VEL
LIN {X 0,Y 502.144,Z 272.832,A -85,B 0,C 180,E1 -5661.954,E2 -5661.954} C_VEL
LIN {X 0,Y 502.235,Z 270.281,A -85,B 0,C 180,E1 -5663.482,E2 -5663.482} C_VEL
LIN {X 0,Y 502.247,Z 266.926,A -85,B 0,C 180,E1 -5664.781,E2 -5664.781} C_VEL
LIN {X 0,Y 502.416,Z 262.71,A -85,B 0,C 180,E1 -5665.989,E2 -5665.989} C_VEL
LIN {X 0,Y 502.518,Z 256.357,A -85,B 0,C 180,E1 -5667.395,E2 -5667.395} C_VEL
LIN {X 0,Y 502.812,Z 249.394,A -85,B 0,C 180,E1 -5668.598,E2 -5668.598} C_VEL
LIN {X 0,Y 503.078,Z 240.736,A -85,B 0,C 180,E1 -5669.8,E2 -5669.8} C_VEL
LIN {X 0,Y 503.36,Z 231.888,A -85,B 0,C 180,E1 -5670.8,E2 -5670.8} C_VEL
LIN {X 0,Y 503.742,Z 222.153,A -85,B 0,C 180,E1 -5671.699,E2 -5671.699} C_VEL
LIN {X 0,Y 504.105,Z 211.397,A -85,B 0,C 180,E1 -5672.497,E2 -5672.497} C_VEL
LIN {X 0,Y 504.436,Z 199.389,A -85,B 0,C 180,E1 -5673.195,E2 -5673.195} C_VEL
LIN {X 0,Y 504.675,Z 186.846,A -85,B 0,C 180,E1 -5673.743,E2 -5673.743} C_VEL
LIN {X 0,Y 504.858,Z 174.381,A -85,B 0,C 180,E1 -5674.116,E2 -5674.116} C_VEL
LIN {X 0,Y 505.033,Z 156.815,A -85,B 0,C 180,E1 -5674.415,E2 -5674.415} C_VEL
LIN {X 0,Y 505.396,Z 74.311,A -85,B 0,C 180,E1 -5675.594,E2 -5675.594} C_VEL
LIN {X 0,Y 503.347,Z 64.16,A -85,B 0,C 180,E1 -5675.81,E2 -5675.81} C_VEL
LIN {X 0,Y 503.563,Z 54.912,A -85,B 0,C 180,E1 -5677.729,E2 -5677.729} C_VEL
LIN {X 0,Y 502.871,Z 49.85,A -85,B 0,C 180,E1 -5678.843,E2 -5678.843} C_VEL
LIN {X 0,Y 502.848,Z 49.845,A -85,B 0,C 180,E1 -5682.102,E2 -5682.102} C_VEL
LIN {X 0,Y 502.851,Z 49.843,A -85,B 0,C 180,E1 -5685.4,E2 -5685.4} C_VEL
LIN {X 0,Y 502.843,Z 49.848,A -85,B 0,C 180,E1 -5688.12,E2 -5688.12} C_VEL
LIN {X 0,Y 502.831,Z 49.851,A -85,B 0,C 180,E1 -5690.536,E2 -5690.536} C_VEL
LIN {X 0,Y 502.79,Z 49.851,A -85,B 0,C 180,E1 -5693.041,E2 -5693.041} C_VEL
LIN {X 0,Y 502.824,Z 49.849,A -85,B 0,C 180,E1 -5695.677,E2 -5695.677} C_VEL
LIN {X 0,Y 502.843,Z 49.848,A -85,B 0,C 180,E1 -5698.373,E2 -5698.373} C_VEL
LIN {X 0,Y 502.795,Z 49.852,A -85,B 0,C 180,E1 -5701.499,E2 -5701.499} C_VEL
LIN {X 0,Y 502.807,Z 49.85,A -85,B 0,C 180,E1 -5704.445,E2 -5704.445} C_VEL
LIN {X 0,Y 502.783,Z 49.853,A -85,B 0,C 180,E1 -5707.178,E2 -5707.178} C_VEL
LIN {X 0,Y 502.79,Z 49.854,A -85,B 0,C 180,E1 -5710.015,E2 -5710.015} C_VEL
LIN {X 0,Y 502.806,Z 49.85,A -85,B 0,C 180,E1 -5712.199,E2 -5712.199} C_VEL
LIN {X 0,Y 502.789,Z 49.859,A -85,B 0,C 180,E1 -5715.47,E2 -5715.47} C_VEL
LIN {X 0,Y 502.823,Z 49.85,A -85,B 0,C 180,E1 -5718.934,E2 -5718.934} C_VEL
LIN {X 0,Y 502.796,Z 49.85,A -85,B 0,C 180,E1 -5722.046,E2 -5722.046} C_VEL
LIN {X 0,Y 502.805,Z 49.856,A -85,B 0,C 180,E1 -5725.035,E2 -5725.035} C_VEL
LIN {X 0,Y 502.787,Z 49.851,A -85,B 0,C 180,E1 -5727.916,E2 -5727.916} C_VEL
LIN {X 0,Y 502.828,Z 49.852,A -85,B 0,C 180,E1 -5730.713,E2 -5730.713} C_VEL
LIN {X 0,Y 502.867,Z 49.842,A -85,B 0,C 180,E1 -5733.44,E2 -5733.44} C_VEL
LIN {X 0,Y 502.783,Z 49.853,A -85,B 0,C 180,E1 -5736.086,E2 -5736.086} C_VEL
LIN {X 0,Y 502.788,Z 49.858,A -85,B 0,C 180,E1 -5738.689,E2 -5738.689} C_VEL
LIN {X 0,Y 502.828,Z 49.847,A -85,B 0,C 180,E1 -5741.248,E2 -5741.248} C_VEL
LIN {X 0,Y 502.854,Z 49.848,A -85,B 0,C 180,E1 -5744.601,E2 -5744.601} C_VEL
LIN {X 0,Y 502.882,Z 49.844,A -85,B 0,C 180,E1 -5748.039,E2 -5748.039} C_VEL
LIN {X 0,Y 502.87,Z 49.841,A -85,B 0,C 180,E1 -5751.157,E2 -5751.157} C_VEL
LIN {X 0,Y 502.917,Z 49.837,A -85,B 0,C 180,E1 -5753.581,E2 -5753.581} C_VEL
LIN {X 0,Y 502.879,Z 49.84,A -85,B 0,C 180,E1 -5756.795,E2 -5756.795} C_VEL
LIN {X 0,Y 503.039,Z 49.82,A -85,B 0,C 180,E1 -5759.2,E2 -5759.2} C_VEL
LIN {X 0,Y 502.906,Z 49.842,A -85,B 0,C 180,E1 -5761.602,E2 -5761.602} C_VEL
LIN {X 0,Y 502.9,Z 49.839,A -85,B 0,C 180,E1 -5763.205,E2 -5763.205} C_VEL
LIN {X 0,Y 502.882,Z 49.839,A -85,B 0,C 180,E1 -5766.419,E2 -5766.419} C_VEL
LIN {X 0,Y 502.869,Z 49.842,A -85,B 0,C 180,E1 -5768.843,E2 -5768.843} C_VEL
LIN {X 0,Y 502.851,Z 49.844,A -85,B 0,C 180,E1 -5772.102,E2 -5772.102} C_VEL
LIN {X 0,Y 502.854,Z 49.85,A -85,B 0,C 180,E1 -5775.4,E2 -5775.4} C_VEL
LIN {X 0,Y 502.829,Z 49.849,A -85,B 0,C 180,E1 -5778.752,E2 -5778.752} C_VEL
LIN {X 0,Y 502.789,Z 49.856,A -85,B 0,C 180,E1 -5781.311,E2 -5781.311} C_VEL
LIN {X 0,Y 502.779,Z 49.852,A -85,B 0,C 180,E1 -5783.915,E2 -5783.915} C_VEL
LIN {X 0,Y 502.841,Z 49.848,A -85,B 0,C 180,E1 -5786.568,E2 -5786.568} C_VEL
LIN {X 0,Y 502.82,Z 49.847,A -85,B 0,C 180,E1 -5789.935,E2 -5789.935} C_VEL
LIN {X 0,Y 502.834,Z 49.849,A -85,B 0,C 180,E1 -5793.031,E2 -5793.031} C_VEL
LIN {X 0,Y 502.776,Z 49.854,A -85,B 0,C 180,E1 -5795.951,E2 -5795.951} C_VEL
LIN {X 0,Y 502.805,Z 49.851,A -85,B 0,C 180,E1 -5798.976,E2 -5798.976} C_VEL
LIN {X 0,Y 502.799,Z 49.855,A -85,B 0,C 180,E1 -5802.139,E2 -5802.139} C_VEL
LIN {X 0,Y 502.789,Z 49.851,A -85,B 0,C 180,E1 -5805.47,E2 -5805.47} C_VEL
LIN {X 0,Y 502.798,Z 49.854,A -85,B 0,C 180,E1 -5807.86,E2 -5807.86} C_VEL
LIN {X 0,Y 502.8,Z 49.849,A -85,B 0,C 180,E1 -5811.023,E2 -5811.023} C_VEL
LIN {X 0,Y 502.775,Z 49.857,A -85,B 0,C 180,E1 -5814.17,E2 -5814.17} C_VEL
LIN {X 0,Y 502.834,Z 49.845,A -85,B 0,C 180,E1 -5816.994,E2 -5816.994} C_VEL
LIN {X 0,Y 502.818,Z 49.853,A -85,B 0,C 180,E1 -5820.065,E2 -5820.065} C_VEL
LIN {X 0,Y 502.834,Z 49.848,A -85,B 0,C 180,E1 -5822.533,E2 -5822.533} C_VEL
LIN {X 0,Y 502.911,Z 50.02,A -85,B 0,C 180,E1 -5824.245,E2 -5824.245} C_VEL
LIN {X 0,Y 504.58,Z 59.122,A -85,B 0,C 180,E1 -5825.739,E2 -5825.739} C_VEL
LIN {X 0,Y 504.15,Z 75.918,A -85,B 0,C 180,E1 -5828.32,E2 -5828.32} C_VEL
LIN {X 0,Y 503.58,Z 97.717,A -85,B 0,C 180,E1 -5831.625,E2 -5831.625} C_VEL
LIN {X 0,Y 503.159,Z 115.007,A -85,B 0,C 180,E1 -5834.202,E2 -5834.202} C_VEL
LIN {X 0,Y 505.285,Z 130.695,A -85,B 0,C 180,E1 -5834.491,E2 -5834.491} C_VEL
LIN {X 0,Y 504.764,Z 224.253,A -85,B 0,C 180,E1 -5835.846,E2 -5835.846} C_VEL
LIN {X 0,Y 504.484,Z 237.356,A -85,B 0,C 180,E1 -5836.198,E2 -5836.198} C_VEL
LIN {X 0,Y 504.152,Z 250.016,A -85,B 0,C 180,E1 -5836.702,E2 -5836.702} C_VEL
LIN {X 0,Y 503.815,Z 261.336,A -85,B 0,C 180,E1 -5837.312,E2 -5837.312} C_VEL
LIN {X 0,Y 503.389,Z 272.949,A -85,B 0,C 180,E1 -5838.116,E2 -5838.116} C_VEL
LIN {X 0,Y 503.083,Z 283.464,A -85,B 0,C 180,E1 -5839.027,E2 -5839.027} C_VEL
LIN {X 0,Y 502.78,Z 292.053,A -85,B 0,C 180,E1 -5839.937,E2 -5839.937} C_VEL
LIN {X 0,Y 502.528,Z 299.98,A -85,B 0,C 180,E1 -5840.948,E2 -5840.948} C_VEL
LIN {X 0,Y 502.355,Z 307.728,A -85,B 0,C 180,E1 -5842.16,E2 -5842.16} C_VEL
LIN {X 0,Y 502.187,Z 314.866,A -85,B 0,C 180,E1 -5843.572,E2 -5843.572} C_VEL
LIN {X 0,Y 502.168,Z 319.62,A -85,B 0,C 180,E1 -5844.781,E2 -5844.781} C_VEL
LIN {X 0,Y 502.164,Z 323.251,A -85,B 0,C 180,E1 -5845.987,E2 -5845.987} C_VEL
LIN {X 0,Y 502.158,Z 325.123,A -85,B 0,C 180,E1 -5846.791,E2 -5846.791} C_VEL
LIN {X 0,Y 502.128,Z 326.525,A -85,B 0,C 180,E1 -5847.593,E2 -5847.593} C_VEL
LIN {X 0,Y 502.016,Z 328.128,A -85,B 0,C 180,E1 -5849.198,E2 -5849.198} C_VEL
LIN {X 0,Y 502.017,Z 328.344,A -85,B 0,C 180,E1 -5850,E2 -5850} C_VEL
LIN {X 0,Y 502.044,Z 327.51,A -85,B 0,C 180,E1 -5851.604,E2 -5851.604} C_VEL
LIN {X 0,Y 502.128,Z 326.509,A -85,B 0,C 180,E1 -5852.406,E2 -5852.406} C_VEL
LIN {X 0,Y 502.158,Z 325.102,A -85,B 0,C 180,E1 -5853.209,E2 -5853.209} C_VEL
LIN {X 0,Y 502.102,Z 322.138,A -85,B 0,C 180,E1 -5854.415,E2 -5854.415} C_VEL
LIN {X 0,Y 502.183,Z 318.137,A -85,B 0,C 180,E1 -5855.622,E2 -5855.622} C_VEL
LIN {X 0,Y 502.272,Z 312.086,A -85,B 0,C 180,E1 -5857.012,E2 -5857.012} C_VEL
LIN {X 0,Y 502.414,Z 305.266,A -85,B 0,C 180,E1 -5858.244,E2 -5858.244} C_VEL
LIN {X 0,Y 502.634,Z 296.936,A -85,B 0,C 180,E1 -5859.456,E2 -5859.456} C_VEL
LIN {X 0,Y 502.924,Z 288.412,A -85,B 0,C 180,E1 -5860.467,E2 -5860.467} C_VEL
LIN {X 0,Y 503.297,Z 277.893,A -85,B 0,C 180,E1 -5861.478,E2 -5861.478} C_VEL
LIN {X 0,Y 503.614,Z 266.63,A -85,B 0,C 180,E1 -5862.349,E2 -5862.349} C_VEL
LIN {X 0,Y 504.02,Z 254.189,A -85,B 0,C 180,E1 -5863.096,E2 -5863.096} C_VEL
LIN {X 0,Y 504.378,Z 241.856,A -85,B 0,C 180,E1 -5863.651,E2 -5863.651} C_VEL
LIN {X 0,Y 504.682,Z 229.247,A -85,B 0,C 180,E1 -5864.054,E2 -5864.054} C_VEL
LIN {X 0,Y 504.905,Z 216.235,A -85,B 0,C 180,E1 -5864.304,E2 -5864.304} C_VEL
LIN {X 0,Y 505.211,Z 129.018,A -85,B 0,C 180,E1 -5865.558,E2 -5865.558} C_VEL
LIN {X 0,Y 503.185,Z 114.677,A -85,B 0,C 180,E1 -5865.837,E2 -5865.837} C_VEL
LIN {X 0,Y 503.735,Z 94.253,A -85,B 0,C 180,E1 -5868.928,E2 -5868.928} C_VEL
LIN {X 0,Y 504.229,Z 76.365,A -85,B 0,C 180,E1 -5871.676,E2 -5871.676} C_VEL
LIN {X 0,Y 504.748,Z 59.869,A -85,B 0,C 180,E1 -5874.252,E2 -5874.252} C_VEL
LIN {X 0,Y 502.876,Z 49.847,A -85,B 0,C 180,E1 -5875.98,E2 -5875.98} C_VEL
LIN {X 0,Y 502.827,Z 49.848,A -85,B 0,C 180,E1 -5879.288,E2 -5879.288} C_VEL
LIN {X 0,Y 502.785,Z 49.859,A -85,B 0,C 180,E1 -5882.085,E2 -5882.085} C_VEL
LIN {X 0,Y 502.799,Z 49.851,A -85,B 0,C 180,E1 -5884.966,E2 -5884.966} C_VEL
LIN {X 0,Y 502.796,Z 49.857,A -85,B 0,C 180,E1 -5887.954,E2 -5887.954} C_VEL
LIN {X 0,Y 502.823,Z 49.848,A -85,B 0,C 180,E1 -5891.066,E2 -5891.066} C_VEL
LIN {X 0,Y 502.789,Z 49.849,A -85,B 0,C 180,E1 -5894.53,E2 -5894.53} C_VEL
LIN {X 0,Y 502.798,Z 49.853,A -85,B 0,C 180,E1 -5897.861,E2 -5897.861} C_VEL
LIN {X 0,Y 502.805,Z 49.85,A -85,B 0,C 180,E1 -5901.024,E2 -5901.024} C_VEL
LIN {X 0,Y 502.778,Z 49.852,A -85,B 0,C 180,E1 -5904.169,E2 -5904.169} C_VEL
LIN {X 0,Y 502.834,Z 49.849,A -85,B 0,C 180,E1 -5906.994,E2 -5906.994} C_VEL
LIN {X 0,Y 502.819,Z 49.845,A -85,B 0,C 180,E1 -5910.065,E2 -5910.065} C_VEL
LIN {X 0,Y 502.837,Z 49.849,A -85,B 0,C 180,E1 -5912.533,E2 -5912.533} C_VEL
LIN {X 0,Y 502.827,Z 49.849,A -85,B 0,C 180,E1 -5915.3,E2 -5915.3} C_VEL
LIN {X 0,Y 502.784,Z 49.85,A -85,B 0,C 180,E1 -5917.826,E2 -5917.826} C_VEL
LIN {X 0,Y 502.826,Z 49.851,A -85,B 0,C 180,E1 -5920.4,E2 -5920.4} C_VEL
LIN {X 0,Y 502.833,Z 49.846,A -85,B 0,C 180,E1 -5922.931,E2 -5922.931} C_VEL
LIN {X 0,Y 502.85,Z 49.844,A -85,B 0,C 180,E1 -5925.429,E2 -5925.429} C_VEL
LIN {X 0,Y 502.882,Z 49.842,A -85,B 0,C 180,E1 -5928.717,E2 -5928.717} C_VEL
LIN {X 0,Y 502.906,Z 49.842,A -85,B 0,C 180,E1 -5931.967,E2 -5931.967} C_VEL
LIN {X 0,Y 502.939,Z 49.836,A -85,B 0,C 180,E1 -5934.386,E2 -5934.386} C_VEL
LIN {X 0,Y 503.024,Z 49.825,A -85,B 0,C 180,E1 -5937.598,E2 -5937.598} C_VEL
LIN {X 0,Y 503.032,Z 49.827,A -85,B 0,C 180,E1 -5940,E2 -5940} C_VEL
LIN {X 0,Y 503.027,Z 49.821,A -85,B 0,C 180,E1 -5942.402,E2 -5942.402} C_VEL
LIN {X 0,Y 502.926,Z 49.841,A -85,B 0,C 180,E1 -5945.614,E2 -5945.614} C_VEL
LIN {X 0,Y 502.885,Z 49.838,A -85,B 0,C 180,E1 -5948.034,E2 -5948.034} C_VEL
LIN {X 0,Y 502.881,Z 49.847,A -85,B 0,C 180,E1 -5951.283,E2 -5951.283} C_VEL
LIN {X 0,Y 502.848,Z 49.842,A -85,B 0,C 180,E1 -5954.571,E2 -5954.571} C_VEL
LIN {X 0,Y 502.821,Z 49.846,A -85,B 0,C 180,E1 -5957.908,E2 -5957.908} C_VEL
LIN {X 0,Y 502.833,Z 49.848,A -85,B 0,C 180,E1 -5960.536,E2 -5960.536} C_VEL
LIN {X 0,Y 502.794,Z 49.855,A -85,B 0,C 180,E1 -5963.04,E2 -5963.04} C_VEL
LIN {X 0,Y 502.809,Z 49.849,A -85,B 0,C 180,E1 -5965.677,E2 -5965.677} C_VEL
LIN {X 0,Y 502.799,Z 49.853,A -85,B 0,C 180,E1 -5968.375,E2 -5968.375} C_VEL
LIN {X 0,Y 502.799,Z 49.851,A -85,B 0,C 180,E1 -5971.143,E2 -5971.143} C_VEL
LIN {X 0,Y 502.791,Z 49.853,A -85,B 0,C 180,E1 -5973.995,E2 -5973.995} C_VEL
LIN {X 0,Y 502.767,Z 49.854,A -85,B 0,C 180,E1 -5977.176,E2 -5977.176} C_VEL
LIN {X 0,Y 502.786,Z 49.856,A -85,B 0,C 180,E1 -5980.015,E2 -5980.015} C_VEL
LIN {X 0,Y 502.805,Z 49.855,A -85,B 0,C 180,E1 -5982.199,E2 -5982.199} C_VEL
LIN {X 0,Y 502.787,Z 49.855,A -85,B 0,C 180,E1 -5985.47,E2 -5985.47} C_VEL
LIN {X 0,Y 502.796,Z 49.858,A -85,B 0,C 180,E1 -5987.86,E2 -5987.86} C_VEL
LIN {X 0,Y 502.795,Z 49.852,A -85,B 0,C 180,E1 -5991.023,E2 -5991.023} C_VEL
LIN {X 0,Y 502.772,Z 49.858,A -85,B 0,C 180,E1 -5994.17,E2 -5994.17} C_VEL
LIN {X 0,Y 502.808,Z 49.854,A -85,B 0,C 180,E1 -5997.213,E2 -5997.213} C_VEL
LIN {X 0,Y 502.115,Z 49.944,A -85,B 0,C 180,E1 -5997.881,E2 -5997.881} C_VEL
LIN {X 0,Y 499.281,Z 50.297,A -85,B 0,C 180,E1 -5998.967,E2 -5998.967} C_VEL
LIN {X 0,Y 496.902,Z 50.593,A -85,B 0,C 180,E1 -5999.842,E2 -5999.842} C_VEL
LIN {X 0,Y 495.876,Z 50.72,A -85,B 0,C 180,E1 -6000.518,E2 -6000.518} C_VEL
LIN {X 0,Y 495.788,Z 50.731,A -85,B 0,C 180,E1 -6000.746,E2 -6000.746} C_VEL
LIN {X 0,Y 495.827,Z 50.944,A -85,B 0,C 180,E1 -6001.015,E2 -6001.015} C_VEL
LIN {X 0,Y 496.594,Z 56.066,A -85,B 0,C 180,E1 -6002.158,E2 -6002.158} C_VEL
LIN {X 0,Y 496.505,Z 64.78,A -85,B 0,C 180,E1 -6003.997,E2 -6003.997} C_VEL
LIN {X 0,Y 498.808,Z 76.592,A -85,B 0,C 180,E1 -6004.257,E2 -6004.257} C_VEL
LIN {X 0,Y 498.148,Z 171.325,A -85,B 0,C 180,E1 -6005.655,E2 -6005.655} C_VEL
LIN {X 0,Y 497.948,Z 184.949,A -85,B 0,C 180,E1 -6006.033,E2 -6006.033} C_VEL
LIN {X 0,Y 497.721,Z 197.834,A -85,B 0,C 180,E1 -6006.568,E2 -6006.568} C_VEL
LIN {X 0,Y 497.332,Z 209.719,A -85,B 0,C 180,E1 -6007.241,E2 -6007.241} C_VEL
LIN {X 0,Y 496.892,Z 221.44,A -85,B 0,C 180,E1 -6008.096,E2 -6008.096} C_VEL
LIN {X 0,Y 496.559,Z 232.124,A -85,B 0,C 180,E1 -6009.087,E2 -6009.087} C_VEL
LIN {X 0,Y 496.171,Z 241.189,A -85,B 0,C 180,E1 -6010.126,E2 -6010.126} C_VEL
LIN {X 0,Y 495.859,Z 248.948,A -85,B 0,C 180,E1 -6011.211,E2 -6011.211} C_VEL
LIN {X 0,Y 495.629,Z 256.234,A -85,B 0,C 180,E1 -6012.463,E2 -6012.463} C_VEL
LIN {X 0,Y 495.418,Z 261.191,A -85,B 0,C 180,E1 -6013.518,E2 -6013.518} C_VEL
LIN {X 0,Y 495.27,Z 265.968,A -85,B 0,C 180,E1 -6014.783,E2 -6014.783} C_VEL
LIN {X 0,Y 495.15,Z 269.559,A -85,B 0,C 180,E1 -6016.037,E2 -6016.037} C_VEL
LIN {X 0,Y 495.074,Z 271.368,A -85,B 0,C 180,E1 -6016.872,E2 -6016.872} C_VEL
LIN {X 0,Y 495.042,Z 273.531,A -85,B 0,C 180,E1 -6018.4,E2 -6018.4} C_VEL
LIN {X 0,Y 495.029,Z 274.21,A -85,B 0,C 180,E1 -6019.364,E2 -6019.364} C_VEL
LIN {X 0,Y 494.983,Z 274.318,A -85,B 0,C 180,E1 -6020.19,E2 -6020.19} C_VEL
LIN {X 0,Y 495.02,Z 274.026,A -85,B 0,C 180,E1 -6021.015,E2 -6021.015} C_VEL
LIN {X 0,Y 495.119,Z 272.278,A -85,B 0,C 180,E1 -6022.66,E2 -6022.66} C_VEL
LIN {X 0,Y 495.162,Z 270.758,A -85,B 0,C 180,E1 -6023.48,E2 -6023.48} C_VEL
LIN {X 0,Y 495.174,Z 267.715,A -85,B 0,C 180,E1 -6024.707,E2 -6024.707} C_VEL
LIN {X 0,Y 495.336,Z 263.619,A -85,B 0,C 180,E1 -6025.932,E2 -6025.932} C_VEL
LIN {X 0,Y 495.457,Z 257.391,A -85,B 0,C 180,E1 -6027.358,E2 -6027.358} C_VEL
LIN {X 0,Y 495.76,Z 250.605,A -85,B 0,C 180,E1 -6028.578,E2 -6028.578} C_VEL
LIN {X 0,Y 496.044,Z 242.156,A -85,B 0,C 180,E1 -6029.797,E2 -6029.797} C_VEL
LIN {X 0,Y 496.344,Z 233.506,A -85,B 0,C 180,E1 -6030.811,E2 -6030.811} C_VEL
LIN {X 0,Y 496.772,Z 222.863,A -85,B 0,C 180,E1 -6031.824,E2 -6031.824} C_VEL
LIN {X 0,Y 497.159,Z 212.211,A -85,B 0,C 180,E1 -6032.633,E2 -6032.633} C_VEL
LIN {X 0,Y 497.512,Z 200.303,A -85,B 0,C 180,E1 -6033.341,E2 -6033.341} C_VEL
LIN {X 0,Y 497.773,Z 187.914,A -85,B 0,C 180,E1 -6033.896,E2 -6033.896} C_VEL
LIN {X 0,Y 497.962,Z 175.927,A -85,B 0,C 180,E1 -6034.275,E2 -6034.275} C_VEL
LIN {X 0,Y 498.087,Z 160.883,A -85,B 0,C 180,E1 -6034.552,E2 -6034.552} C_VEL
LIN {X 0,Y 498.482,Z 74.893,A -85,B 0,C 180,E1 -6035.799,E2 -6035.799} C_VEL
LIN {X 0,Y 496.362,Z 64.513,A -85,B 0,C 180,E1 -6036.02,E2 -6036.02} C_VEL
LIN {X 0,Y 496.565,Z 55.948,A -85,B 0,C 180,E1 -6037.809,E2 -6037.809} C_VEL
LIN {X 0,Y 495.84,Z 50.726,A -85,B 0,C 180,E1 -6038.97,E2 -6038.97} C_VEL
LIN {X 0,Y 495.83,Z 50.719,A -85,B 0,C 180,E1 -6042.035,E2 -6042.035} C_VEL
LIN {X 0,Y 495.826,Z 50.718,A -85,B 0,C 180,E1 -6045.452,E2 -6045.452} C_VEL
LIN {X 0,Y 495.809,Z 50.726,A -85,B 0,C 180,E1 -6048.247,E2 -6048.247} C_VEL
LIN {X 0,Y 495.776,Z 50.727,A -85,B 0,C 180,E1 -6050.757,E2 -6050.757} C_VEL
LIN {X 0,Y 495.745,Z 50.728,A -85,B 0,C 180,E1 -6053.388,E2 -6053.388} C_VEL
LIN {X 0,Y 495.826,Z 50.719,A -85,B 0,C 180,E1 -6056.749,E2 -6056.749} C_VEL
LIN {X 0,Y 495.769,Z 50.73,A -85,B 0,C 180,E1 -6059.747,E2 -6059.747} C_VEL
LIN {X 0,Y 495.77,Z 50.726,A -85,B 0,C 180,E1 -6062.595,E2 -6062.595} C_VEL
LIN {X 0,Y 495.758,Z 50.731,A -85,B 0,C 180,E1 -6065.537,E2 -6065.537} C_VEL
LIN {X 0,Y 495.766,Z 50.726,A -85,B 0,C 180,E1 -6068.768,E2 -6068.768} C_VEL
LIN {X 0,Y 495.758,Z 50.732,A -85,B 0,C 180,E1 -6071.781,E2 -6071.781} C_VEL
LIN {X 0,Y 495.74,Z 50.733,A -85,B 0,C 180,E1 -6075.141,E2 -6075.141} C_VEL
LIN {X 0,Y 495.759,Z 50.727,A -85,B 0,C 180,E1 -6078.219,E2 -6078.219} C_VEL
LIN {X 0,Y 495.754,Z 50.733,A -85,B 0,C 180,E1 -6081.409,E2 -6081.409} C_VEL
LIN {X 0,Y 495.753,Z 50.728,A -85,B 0,C 180,E1 -6084.463,E2 -6084.463} C_VEL
LIN {X 0,Y 495.771,Z 50.728,A -85,B 0,C 180,E1 -6087.406,E2 -6087.406} C_VEL
LIN {X 0,Y 495.771,Z 50.726,A -85,B 0,C 180,E1 -6090.254,E2 -6090.254} C_VEL
LIN {X 0,Y 495.828,Z 50.721,A -85,B 0,C 180,E1 -6093.251,E2 -6093.251} C_VEL
LIN {X 0,Y 495.747,Z 50.728,A -85,B 0,C 180,E1 -6095.725,E2 -6095.725} C_VEL
LIN {X 0,Y 495.747,Z 50.733,A -85,B 0,C 180,E1 -6098.371,E2 -6098.371} C_VEL
LIN {X 0,Y 495.784,Z 50.726,A -85,B 0,C 180,E1 -6100.972,E2 -6100.972} C_VEL
LIN {X 0,Y 495.829,Z 50.724,A -85,B 0,C 180,E1 -6104.549,E2 -6104.549} C_VEL
LIN {X 0,Y 495.834,Z 50.721,A -85,B 0,C 180,E1 -6107.965,E2 -6107.965} C_VEL
LIN {X 0,Y 495.84,Z 50.717,A -85,B 0,C 180,E1 -6111.03,E2 -6111.03} C_VEL
LIN {X 0,Y 495.871,Z 50.714,A -85,B 0,C 180,E1 -6113.49,E2 -6113.49} C_VEL
LIN {X 0,Y 495.824,Z 50.719,A -85,B 0,C 180,E1 -6116.75,E2 -6116.75} C_VEL
LIN {X 0,Y 495.874,Z 50.715,A -85,B 0,C 180,E1 -6118.376,E2 -6118.376} C_VEL
LIN {X 0,Y 495.988,Z 50.698,A -85,B 0,C 180,E1 -6120.812,E2 -6120.812} C_VEL
LIN {X 0,Y 495.997,Z 50.698,A -85,B 0,C 180,E1 -6122.436,E2 -6122.436} C_VEL
LIN {X 0,Y 495.88,Z 50.719,A -85,B 0,C 180,E1 -6125.694,E2 -6125.694} C_VEL
LIN {X 0,Y 495.839,Z 50.718,A -85,B 0,C 180,E1 -6128.97,E2 -6128.97} C_VEL
LIN {X 0,Y 495.834,Z 50.718,A -85,B 0,C 180,E1 -6132.035,E2 -6132.035} C_VEL
LIN {X 0,Y 495.83,Z 50.724,A -85,B 0,C 180,E1 -6135.452,E2 -6135.452} C_VEL
LIN {X 0,Y 495.78,Z 50.724,A -85,B 0,C 180,E1 -6138.236,E2 -6138.236} C_VEL
LIN {X 0,Y 495.78,Z 50.728,A -85,B 0,C 180,E1 -6140.756,E2 -6140.756} C_VEL
LIN {X 0,Y 495.747,Z 50.731,A -85,B 0,C 180,E1 -6143.387,E2 -6143.387} C_VEL
LIN {X 0,Y 495.767,Z 50.726,A -85,B 0,C 180,E1 -6146.069,E2 -6146.069} C_VEL
LIN {X 0,Y 495.752,Z 50.736,A -85,B 0,C 180,E1 -6148.816,E2 -6148.816} C_VEL
LIN {X 0,Y 495.76,Z 50.726,A -85,B 0,C 180,E1 -6151.725,E2 -6151.725} C_VEL
LIN {X 0,Y 495.766,Z 50.733,A -85,B 0,C 180,E1 -6154.693,E2 -6154.693} C_VEL
LIN {X 0,Y 495.732,Z 50.73,A -85,B 0,C 180,E1 -6157.562,E2 -6157.562} C_VEL
LIN {X 0,Y 495.77,Z 50.729,A -85,B 0,C 180,E1 -6160.7,E2 -6160.7} C_VEL
LIN {X 0,Y 495.732,Z 50.735,A -85,B 0,C 180,E1 -6164.001,E2 -6164.001} C_VEL
LIN {X 0,Y 495.719,Z 50.731,A -85,B 0,C 180,E1 -6167.116,E2 -6167.116} C_VEL
LIN {X 0,Y 495.759,Z 50.734,A -85,B 0,C 180,E1 -6169.953,E2 -6169.953} C_VEL
LIN {X 0,Y 495.722,Z 50.732,A -85,B 0,C 180,E1 -6172.555,E2 -6172.555} C_VEL
LIN {X 0,Y 495.774,Z 50.728,A -85,B 0,C 180,E1 -6175.456,E2 -6175.456} C_VEL
LIN {X 0,Y 495.758,Z 50.728,A -85,B 0,C 180,E1 -6178.364,E2 -6178.364} C_VEL
LIN {X 0,Y 495.79,Z 50.73,A -85,B 0,C 180,E1 -6181.507,E2 -6181.507} C_VEL
LIN {X 0,Y 495.841,Z 50.783,A -85,B 0,C 180,E1 -6184.059,E2 -6184.059} C_VEL
LIN {X 0,Y 497.591,Z 60.007,A -85,B 0,C 180,E1 -6185.598,E2 -6185.598} C_VEL
LIN {X 0,Y 497.296,Z 72.624,A -85,B 0,C 180,E1 -6187.568,E2 -6187.568} C_VEL
LIN {X 0,Y 496.735,Z 92.158,A -85,B 0,C 180,E1 -6190.58,E2 -6190.58} C_VEL
LIN {X 0,Y 496.302,Z 108.824,A -85,B 0,C 180,E1 -6193.124,E2 -6193.124} C_VEL
LIN {X 0,Y 496.147,Z 114.477,A -85,B 0,C 180,E1 -6193.982,E2 -6193.982} C_VEL
LIN {X 0,Y 498.428,Z 131.925,A -85,B 0,C 180,E1 -6194.308,E2 -6194.308} C_VEL
LIN {X 0,Y 497.881,Z 223.411,A -85,B 0,C 180,E1 -6195.646,E2 -6195.646} C_VEL
LIN {X 0,Y 497.585,Z 236.676,A -85,B 0,C 180,E1 -6196.002,E2 -6196.002} C_VEL
LIN {X 0,Y 497.216,Z 249.422,A -85,B 0,C 180,E1 -6196.513,E2 -6196.513} C_VEL
LIN {X 0,Y 496.834,Z 261.071,A -85,B 0,C 180,E1 -6197.147,E2 -6197.147} C_VEL
LIN {X 0,Y 496.407,Z 272.459,A -85,B 0,C 180,E1 -6197.946,E2 -6197.946} C_VEL
LIN {X 0,Y 496.057,Z 282.999,A -85,B 0,C 180,E1 -6198.87,E2 -6198.87} C_VEL
LIN {X 0,Y 495.749,Z 291.612,A -85,B 0,C 180,E1 -6199.793,E2 -6199.793} C_VEL
LIN {X 0,Y 495.464,Z 299.554,A -85,B 0,C 180,E1 -6200.817,E2 -6200.817} C_VEL
LIN {X 0,Y 495.303,Z 307.319,A -85,B 0,C 180,E1 -6202.048,E2 -6202.048} C_VEL
LIN {X 0,Y 495.107,Z 314.465,A -85,B 0,C 180,E1 -6203.479,E2 -6203.479} C_VEL
LIN {X 0,Y 495.096,Z 319.226,A -85,B 0,C 180,E1 -6204.706,E2 -6204.706} C_VEL
LIN {X 0,Y 495.056,Z 322.86,A -85,B 0,C 180,E1 -6205.93,E2 -6205.93} C_VEL
LIN {X 0,Y 495.077,Z 324.736,A -85,B 0,C 180,E1 -6206.745,E2 -6206.745} C_VEL
LIN {X 0,Y 495.062,Z 326.14,A -85,B 0,C 180,E1 -6207.559,E2 -6207.559} C_VEL
LIN {X 0,Y 494.934,Z 327.744,A -85,B 0,C 180,E1 -6209.186,E2 -6209.186} C_VEL
LIN {X 0,Y 494.933,Z 327.96,A -85,B 0,C 180,E1 -6210,E2 -6210} C_VEL
LIN {X 0,Y 494.97,Z 327.127,A -85,B 0,C 180,E1 -6211.627,E2 -6211.627} C_VEL
LIN {X 0,Y 495.062,Z 326.127,A -85,B 0,C 180,E1 -6212.441,E2 -6212.441} C_VEL
LIN {X 0,Y 495.077,Z 324.72,A -85,B 0,C 180,E1 -6213.255,E2 -6213.255} C_VEL
LIN {X 0,Y 495.008,Z 321.758,A -85,B 0,C 180,E1 -6214.479,E2 -6214.479} C_VEL
LIN {X 0,Y 495.075,Z 317.759,A -85,B 0,C 180,E1 -6215.703,E2 -6215.703} C_VEL
LIN {X 0,Y 495.193,Z 311.615,A -85,B 0,C 180,E1 -6217.134,E2 -6217.134} C_VEL
LIN {X 0,Y 495.339,Z 304.905,A -85,B 0,C 180,E1 -6218.362,E2 -6218.362} C_VEL
LIN {X 0,Y 495.59,Z 296.591,A -85,B 0,C 180,E1 -6219.592,E2 -6219.592} C_VEL
LIN {X 0,Y 495.926,Z 288.089,A -85,B 0,C 180,E1 -6220.616,E2 -6220.616} C_VEL
LIN {X 0,Y 496.328,Z 277.597,A -85,B 0,C 180,E1 -6221.641,E2 -6221.641} C_VEL
LIN {X 0,Y 496.598,Z 267.517,A -85,B 0,C 180,E1 -6222.443,E2 -6222.443} C_VEL
LIN {X 0,Y 497.035,Z 255.886,A -85,B 0,C 180,E1 -6223.18,E2 -6223.18} C_VEL
LIN {X 0,Y 497.383,Z 244.333,A -85,B 0,C 180,E1 -6223.743,E2 -6223.743} C_VEL
LIN {X 0,Y 497.76,Z 231.082,A -85,B 0,C 180,E1 -6224.201,E2 -6224.201} C_VEL
LIN {X 0,Y 498.05,Z 218.234,A -85,B 0,C 180,E1 -6224.479,E2 -6224.479} C_VEL
LIN {X 0,Y 498.424,Z 129.877,A -85,B 0,C 180,E1 -6225.77,E2 -6225.77} C_VEL
LIN {X 0,Y 496.177,Z 114.2,A -85,B 0,C 180,E1 -6226.094,E2 -6226.094} C_VEL
LIN {X 0,Y 496.787,Z 93.99,A -85,B 0,C 180,E1 -6229.203,E2 -6229.203} C_VEL
LIN {X 0,Y 497.289,Z 76.136,A -85,B 0,C 180,E1 -6231.994,E2 -6231.994} C_VEL
LIN {X 0,Y 497.809,Z 61.042,A -85,B 0,C 180,E1 -6234.39,E2 -6234.39} C_VEL
LIN {X 0,Y 495.831,Z 50.726,A -85,B 0,C 180,E1 -6236.219,E2 -6236.219} C_VEL
LIN {X 0,Y 495.774,Z 50.728,A -85,B 0,C 180,E1 -6238.815,E2 -6238.815} C_VEL
LIN {X 0,Y 495.758,Z 50.73,A -85,B 0,C 180,E1 -6241.725,E2 -6241.725} C_VEL
LIN {X 0,Y 495.766,Z 50.729,A -85,B 0,C 180,E1 -6244.693,E2 -6244.693} C_VEL
LIN {X 0,Y 495.732,Z 50.734,A -85,B 0,C 180,E1 -6247.562,E2 -6247.562} C_VEL
LIN {X 0,Y 495.769,Z 50.726,A -85,B 0,C 180,E1 -6250.7,E2 -6250.7} C_VEL
LIN {X 0,Y 495.731,Z 50.732,A -85,B 0,C 180,E1 -6254.002,E2 -6254.002} C_VEL
LIN {X 0,Y 495.728,Z 50.732,A -85,B 0,C 180,E1 -6257.117,E2 -6257.117} C_VEL
LIN {X 0,Y 495.762,Z 50.726,A -85,B 0,C 180,E1 -6259.953,E2 -6259.953} C_VEL
LIN {X 0,Y 495.731,Z 50.729,A -85,B 0,C 180,E1 -6262.553,E2 -6262.553} C_VEL
LIN {X 0,Y 495.775,Z 50.728,A -85,B 0,C 180,E1 -6265.456,E2 -6265.456} C_VEL
LIN {X 0,Y 495.759,Z 50.728,A -85,B 0,C 180,E1 -6268.364,E2 -6268.364} C_VEL
LIN {X 0,Y 495.792,Z 50.725,A -85,B 0,C 180,E1 -6271.507,E2 -6271.507} C_VEL
LIN {X 0,Y 495.794,Z 50.72,A -85,B 0,C 180,E1 -6273.932,E2 -6273.932} C_VEL
LIN {X 0,Y 495.763,Z 50.728,A -85,B 0,C 180,E1 -6277.14,E2 -6277.14} C_VEL
LIN {X 0,Y 495.773,Z 50.726,A -85,B 0,C 180,E1 -6280.11,E2 -6280.11} C_VEL
LIN {X 0,Y 495.785,Z 50.726,A -85,B 0,C 180,E1 -6282.681,E2 -6282.681} C_VEL
LIN {X 0,Y 495.795,Z 50.723,A -85,B 0,C 180,E1 -6285.217,E2 -6285.217} C_VEL
LIN {X 0,Y 495.857,Z 50.719,A -85,B 0,C 180,E1 -6288.555,E2 -6288.555} C_VEL
LIN {X 0,Y 495.877,Z 50.716,A -85,B 0,C 180,E1 -6291.852,E2 -6291.852} C_VEL
LIN {X 0,Y 495.895,Z 50.715,A -85,B 0,C 180,E1 -6294.306,E2 -6294.306} C_VEL
LIN {X 0,Y 495.992,Z 50.701,A -85,B 0,C 180,E1 -6297.564,E2 -6297.564} C_VEL
LIN {X 0,Y 495.987,Z 50.699,A -85,B 0,C 180,E1 -6300.812,E2 -6300.812} C_VEL
LIN {X 0,Y 495.995,Z 50.696,A -85,B 0,C 180,E1 -6302.436,E2 -6302.436} C_VEL
LIN {X 0,Y 495.882,Z 50.719,A -85,B 0,C 180,E1 -6305.694,E2 -6305.694} C_VEL
LIN {X 0,Y 495.84,Z 50.715,A -85,B 0,C 180,E1 -6308.148,E2 -6308.148} C_VEL
LIN {X 0,Y 495.856,Z 50.722,A -85,B 0,C 180,E1 -6311.445,E2 -6311.445} C_VEL
LIN {X 0,Y 495.794,Z 50.722,A -85,B 0,C 180,E1 -6314.783,E2 -6314.783} C_VEL
LIN {X 0,Y 495.764,Z 50.73,A -85,B 0,C 180,E1 -6317.319,E2 -6317.319} C_VEL
LIN {X 0,Y 495.772,Z 50.725,A -85,B 0,C 180,E1 -6319.89,E2 -6319.89} C_VEL
LIN {X 0,Y 495.763,Z 50.731,A -85,B 0,C 180,E1 -6322.86,E2 -6322.86} C_VEL
LIN {X 0,Y 495.767,Z 50.727,A -85,B 0,C 180,E1 -6326.069,E2 -6326.069} C_VEL
LIN {X 0,Y 495.747,Z 50.734,A -85,B 0,C 180,E1 -6328.816,E2 -6328.816} C_VEL
LIN {X 0,Y 495.758,Z 50.727,A -85,B 0,C 180,E1 -6331.725,E2 -6331.725} C_VEL
LIN {X 0,Y 495.763,Z 50.731,A -85,B 0,C 180,E1 -6334.692,E2 -6334.692} C_VEL
LIN {X 0,Y 495.723,Z 50.732,A -85,B 0,C 180,E1 -6337.562,E2 -6337.562} C_VEL
LIN {X 0,Y 495.757,Z 50.731,A -85,B 0,C 180,E1 -6340.046,E2 -6340.046} C_VEL
LIN {X 0,Y 495.718,Z 50.734,A -85,B 0,C 180,E1 -6342.884,E2 -6342.884} C_VEL
LIN {X 0,Y 495.725,Z 50.739,A -85,B 0,C 180,E1 -6345.998,E2 -6345.998} C_VEL
LIN {X 0,Y 495.741,Z 50.731,A -85,B 0,C 180,E1 -6348.709,E2 -6348.709} C_VEL
LIN {X 0,Y 495.747,Z 50.733,A -85,B 0,C 180,E1 -6351.408,E2 -6351.408} C_VEL
LIN {X 0,Y 495.745,Z 50.732,A -85,B 0,C 180,E1 -6354.462,E2 -6354.462} C_VEL
LIN {X 0,Y 495.767,Z 50.735,A -85,B 0,C 180,E1 -6357.405,E2 -6357.405} C_VEL
LIN {X 0,Y 495.788,Z 50.731,A -85,B 0,C 180,E1 -6360.746,E2 -6360.746} C_VEL
LIN {X 0,Y 495.5,Z 51.337,A -85,B 0,C 180,E1 -6361.047,E2 -6361.047} C_VEL
LIN {X 0,Y 493.837,Z 53.999,A -85,B 0,C 180,E1 -6361.571,E2 -6361.571} C_VEL
LIN {X 0,Y 490.262,Z 58.797,A -85,B 0,C 180,E1 -6362.414,E2 -6362.414} C_VEL
LIN {X 0,Y 489.618,Z 60.736,A -85,B 0,C 180,E1 -6362.812,E2 -6362.812} C_VEL
LIN {X 0,Y 489.541,Z 65.045,A -85,B 0,C 180,E1 -6363.731,E2 -6363.731} C_VEL
LIN {X 0,Y 492.043,Z 77.55,A -85,B 0,C 180,E1 -6364.023,E2 -6364.023} C_VEL
LIN {X 0,Y 491.319,Z 171.808,A -85,B 0,C 180,E1 -6365.435,E2 -6365.435} C_VEL
LIN {X 0,Y 491.131,Z 185.4,A -85,B 0,C 180,E1 -6365.819,E2 -6365.819} C_VEL
LIN {X 0,Y 490.891,Z 197.214,A -85,B 0,C 180,E1 -6366.311,E2 -6366.311} C_VEL
LIN {X 0,Y 490.503,Z 208.361,A -85,B 0,C 180,E1 -6366.927,E2 -6366.927} C_VEL
LIN {X 0,Y 490.051,Z 220.167,A -85,B 0,C 180,E1 -6367.774,E2 -6367.774} C_VEL
LIN {X 0,Y 489.661,Z 231.175,A -85,B 0,C 180,E1 -6368.774,E2 -6368.774} C_VEL
LIN {X 0,Y 489.248,Z 240.526,A -85,B 0,C 180,E1 -6369.833,E2 -6369.833} C_VEL
LIN {X 0,Y 488.929,Z 248.32,A -85,B 0,C 180,E1 -6370.912,E2 -6370.912} C_VEL
LIN {X 0,Y 488.608,Z 256.006,A -85,B 0,C 180,E1 -6372.223,E2 -6372.223} C_VEL
LIN {X 0,Y 488.391,Z 260.99,A -85,B 0,C 180,E1 -6373.274,E2 -6373.274} C_VEL
LIN {X 0,Y 488.232,Z 266.295,A -85,B 0,C 180,E1 -6374.677,E2 -6374.677} C_VEL
LIN {X 0,Y 488.112,Z 269.599,A -85,B 0,C 180,E1 -6375.832,E2 -6375.832} C_VEL
LIN {X 0,Y 488.017,Z 271.502,A -85,B 0,C 180,E1 -6376.678,E2 -6376.678} C_VEL
LIN {X 0,Y 487.985,Z 272.921,A -85,B 0,C 180,E1 -6377.524,E2 -6377.524} C_VEL
LIN {X 0,Y 487.967,Z 273.918,A -85,B 0,C 180,E1 -6378.367,E2 -6378.367} C_VEL
LIN {X 0,Y 487.941,Z 274.521,A -85,B 0,C 180,E1 -6379.208,E2 -6379.208} C_VEL
LIN {X 0,Y 487.914,Z 274.725,A -85,B 0,C 180,E1 -6380.046,E2 -6380.046} C_VEL
LIN {X 0,Y 487.934,Z 274.489,A -85,B 0,C 180,E1 -6380.884,E2 -6380.884} C_VEL
LIN {X 0,Y 488.015,Z 272.851,A -85,B 0,C 180,E1 -6382.553,E2 -6382.553} C_VEL
LIN {X 0,Y 488.085,Z 271.214,A -85,B 0,C 180,E1 -6383.484,E2 -6383.484} C_VEL
LIN {X 0,Y 488.121,Z 267.259,A -85,B 0,C 180,E1 -6385.044,E2 -6385.044} C_VEL
LIN {X 0,Y 488.318,Z 262.912,A -85,B 0,C 180,E1 -6386.287,E2 -6386.287} C_VEL
LIN {X 0,Y 488.408,Z 257.412,A -85,B 0,C 180,E1 -6387.526,E2 -6387.526} C_VEL
LIN {X 0,Y 488.752,Z 250.531,A -85,B 0,C 180,E1 -6388.764,E2 -6388.764} C_VEL
LIN {X 0,Y 489.061,Z 241.944,A -85,B 0,C 180,E1 -6390,E2 -6390} C_VEL
LIN {X 0,Y 489.39,Z 233.171,A -85,B 0,C 180,E1 -6391.029,E2 -6391.029} C_VEL
LIN {X 0,Y 489.807,Z 222.364,A -85,B 0,C 180,E1 -6392.056,E2 -6392.056} C_VEL
LIN {X 0,Y 490.251,Z 211.418,A -85,B 0,C 180,E1 -6392.876,E2 -6392.876} C_VEL
LIN {X 0,Y 490.616,Z 199.207,A -85,B 0,C 180,E1 -6393.593,E2 -6393.593} C_VEL
LIN {X 0,Y 490.881,Z 187.625,A -85,B 0,C 180,E1 -6394.105,E2 -6394.105} C_VEL
LIN {X 0,Y 491.078,Z 175.169,A -85,B 0,C 180,E1 -6394.489,E2 -6394.489} C_VEL
LIN {X 0,Y 491.269,Z 157.607,A -85,B 0,C 180,E1 -6394.796,E2 -6394.796} C_VEL
LIN {X 0,Y 491.624,Z 75.68,A -85,B 0,C 180,E1 -6396.001,E2 -6396.001} C_VEL
LIN {X 0,Y 489.389,Z 64.852,A -85,B 0,C 180,E1 -6396.235,E2 -6396.235} C_VEL
LIN {X 0,Y 489.572,Z 56.972,A -85,B 0,C 180,E1 -6397.894,E2 -6397.894} C_VEL
LIN {X 0,Y 488.781,Z 51.605,A -85,B 0,C 180,E1 -6399.101,E2 -6399.101} C_VEL
LIN {X 0,Y 488.791,Z 51.596,A -85,B 0,C 180,E1 -6402.116,E2 -6402.116} C_VEL
LIN {X 0,Y 488.779,Z 51.596,A -85,B 0,C 180,E1 -6405.555,E2 -6405.555} C_VEL
LIN {X 0,Y 488.757,Z 51.607,A -85,B 0,C 180,E1 -6408.442,E2 -6408.442} C_VEL
LIN {X 0,Y 488.709,Z 51.605,A -85,B 0,C 180,E1 -6411.071,E2 -6411.071} C_VEL
LIN {X 0,Y 488.682,Z 51.61,A -85,B 0,C 180,E1 -6413.746,E2 -6413.746} C_VEL
LIN {X 0,Y 488.794,Z 51.594,A -85,B 0,C 180,E1 -6416.944,E2 -6416.944} C_VEL
LIN {X 0,Y 488.712,Z 51.608,A -85,B 0,C 180,E1 -6420.363,E2 -6420.363} C_VEL
LIN {X 0,Y 488.738,Z 51.604,A -85,B 0,C 180,E1 -6423.485,E2 -6423.485} C_VEL
LIN {X 0,Y 488.69,Z 51.609,A -85,B 0,C 180,E1 -6426.356,E2 -6426.356} C_VEL
LIN {X 0,Y 488.703,Z 51.608,A -85,B 0,C 180,E1 -6429.255,E2 -6429.255} C_VEL
LIN {X 0,Y 488.71,Z 51.613,A -85,B 0,C 180,E1 -6431.6,E2 -6431.6} C_VEL
LIN {X 0,Y 488.704,Z 51.606,A -85,B 0,C 180,E1 -6434.803,E2 -6434.803} C_VEL
LIN {X 0,Y 488.695,Z 51.614,A -85,B 0,C 180,E1 -6437.475,E2 -6437.475} C_VEL
LIN {X 0,Y 488.736,Z 51.605,A -85,B 0,C 180,E1 -6439.677,E2 -6439.677} C_VEL
LIN {X 0,Y 488.683,Z 51.612,A -85,B 0,C 180,E1 -6442.841,E2 -6442.841} C_VEL
LIN {X 0,Y 488.735,Z 51.602,A -85,B 0,C 180,E1 -6445.888,E2 -6445.888} C_VEL
LIN {X 0,Y 488.696,Z 51.612,A -85,B 0,C 180,E1 -6448.821,E2 -6448.821} C_VEL
LIN {X 0,Y 488.749,Z 51.6,A -85,B 0,C 180,E1 -6451.672,E2 -6451.672} C_VEL
LIN {X 0,Y 488.75,Z 51.603,A -85,B 0,C 180,E1 -6454.445,E2 -6454.445} C_VEL
LIN {X 0,Y 488.727,Z 51.605,A -85,B 0,C 180,E1 -6457.153,E2 -6457.153} C_VEL
LIN {X 0,Y 488.729,Z 51.603,A -85,B 0,C 180,E1 -6459.811,E2 -6459.811} C_VEL
LIN {X 0,Y 488.715,Z 51.611,A -85,B 0,C 180,E1 -6462.423,E2 -6462.423} C_VEL
LIN {X 0,Y 488.767,Z 51.599,A -85,B 0,C 180,E1 -6465,E2 -6465} C_VEL
LIN {X 0,Y 488.811,Z 51.599,A -85,B 0,C 180,E1 -6468.388,E2 -6468.388} C_VEL
LIN {X 0,Y 488.79,Z 51.597,A -85,B 0,C 180,E1 -6471.733,E2 -6471.733} C_VEL
LIN {X 0,Y 488.855,Z 51.593,A -85,B 0,C 180,E1 -6474.224,E2 -6474.224} C_VEL
LIN {X 0,Y 488.96,Z 51.576,A -85,B 0,C 180,E1 -6477.529,E2 -6477.529} C_VEL
LIN {X 0,Y 488.939,Z 51.576,A -85,B 0,C 180,E1 -6480.824,E2 -6480.824} C_VEL
LIN {X 0,Y 488.965,Z 51.574,A -85,B 0,C 180,E1 -6482.471,E2 -6482.471} C_VEL
LIN {X 0,Y 488.837,Z 51.595,A -85,B 0,C 180,E1 -6485.776,E2 -6485.776} C_VEL
LIN {X 0,Y 488.79,Z 51.595,A -85,B 0,C 180,E1 -6488.267,E2 -6488.267} C_VEL
LIN {X 0,Y 488.811,Z 51.598,A -85,B 0,C 180,E1 -6491.612,E2 -6491.612} C_VEL
LIN {X 0,Y 488.767,Z 51.602,A -85,B 0,C 180,E1 -6495,E2 -6495} C_VEL
LIN {X 0,Y 488.751,Z 51.6,A -85,B 0,C 180,E1 -6498.442,E2 -6498.442} C_VEL
LIN {X 0,Y 488.712,Z 51.613,A -85,B 0,C 180,E1 -6501.071,E2 -6501.071} C_VEL
LIN {X 0,Y 488.68,Z 51.609,A -85,B 0,C 180,E1 -6503.746,E2 -6503.746} C_VEL
LIN {X 0,Y 488.724,Z 51.606,A -85,B 0,C 180,E1 -6506.474,E2 -6506.474} C_VEL
LIN {X 0,Y 488.716,Z 51.606,A -85,B 0,C 180,E1 -6509.271,E2 -6509.271} C_VEL
LIN {X 0,Y 488.707,Z 51.607,A -85,B 0,C 180,E1 -6512.147,E2 -6512.147} C_VEL
LIN {X 0,Y 488.718,Z 51.605,A -85,B 0,C 180,E1 -6515.115,E2 -6515.115} C_VEL
LIN {X 0,Y 488.683,Z 51.612,A -85,B 0,C 180,E1 -6518.2,E2 -6518.2} C_VEL
LIN {X 0,Y 488.722,Z 51.611,A -85,B 0,C 180,E1 -6520.345,E2 -6520.345} C_VEL
LIN {X 0,Y 488.688,Z 51.609,A -85,B 0,C 180,E1 -6523.655,E2 -6523.655} C_VEL
LIN {X 0,Y 488.68,Z 51.614,A -85,B 0,C 180,E1 -6526.344,E2 -6526.344} C_VEL
LIN {X 0,Y 488.706,Z 51.608,A -85,B 0,C 180,E1 -6529.673,E2 -6529.673} C_VEL
LIN {X 0,Y 488.673,Z 51.609,A -85,B 0,C 180,E1 -6532.84,E2 -6532.84} C_VEL
LIN {X 0,Y 488.727,Z 51.61,A -85,B 0,C 180,E1 -6535.887,E2 -6535.887} C_VEL
LIN {X 0,Y 488.694,Z 51.607,A -85,B 0,C 180,E1 -6538.82,E2 -6538.82} C_VEL
LIN {X 0,Y 488.747,Z 51.608,A -85,B 0,C 180,E1 -6541.671,E2 -6541.671} C_VEL
LIN {X 0,Y 488.809,Z 51.741,A -85,B 0,C 180,E1 -6543.904,E2 -6543.904} C_VEL
LIN {X 0,Y 490.581,Z 60.874,A -85,B 0,C 180,E1 -6545.452,E2 -6545.452} C_VEL
LIN {X 0,Y 490.436,Z 70.841,A -85,B 0,C 180,E1 -6547.036,E2 -6547.036} C_VEL
LIN {X 0,Y 489.764,Z 91.652,A -85,B 0,C 180,E1 -6550.292,E2 -6550.292} C_VEL
LIN {X 0,Y 489.29,Z 108.329,A -85,B 0,C 180,E1 -6552.875,E2 -6552.875} C_VEL
LIN {X 0,Y 489.132,Z 114.166,A -85,B 0,C 180,E1 -6553.767,E2 -6553.767} C_VEL
LIN {X 0,Y 491.545,Z 131.781,A -85,B 0,C 180,E1 -6554.101,E2 -6554.101} C_VEL
LIN {X 0,Y 490.983,Z 223.542,A -85,B 0,C 180,E1 -6555.466,E2 -6555.466} C_VEL
LIN {X 0,Y 490.7,Z 235.881,A -85,B 0,C 180,E1 -6555.802,E2 -6555.802} C_VEL
LIN {X 0,Y 490.286,Z 248.74,A -85,B 0,C 180,E1 -6556.319,E2 -6556.319} C_VEL
LIN {X 0,Y 489.88,Z 260.486,A -85,B 0,C 180,E1 -6556.962,E2 -6556.962} C_VEL
LIN {X 0,Y 489.435,Z 271.974,A -85,B 0,C 180,E1 -6557.776,E2 -6557.776} C_VEL
LIN {X 0,Y 489.066,Z 282.493,A -85,B 0,C 180,E1 -6558.709,E2 -6558.709} C_VEL
LIN {X 0,Y 488.701,Z 291.131,A -85,B 0,C 180,E1 -6559.644,E2 -6559.644} C_VEL
LIN {X 0,Y 488.425,Z 299.096,A -85,B 0,C 180,E1 -6560.684,E2 -6560.684} C_VEL
LIN {X 0,Y 488.228,Z 306.883,A -85,B 0,C 180,E1 -6561.932,E2 -6561.932} C_VEL
LIN {X 0,Y 488.036,Z 314.044,A -85,B 0,C 180,E1 -6563.384,E2 -6563.384} C_VEL
LIN {X 0,Y 488.001,Z 318.814,A -85,B 0,C 180,E1 -6564.629,E2 -6564.629} C_VEL
LIN {X 0,Y 487.95,Z 322.456,A -85,B 0,C 180,E1 -6565.87,E2 -6565.87} C_VEL
LIN {X 0,Y 487.997,Z 324.339,A -85,B 0,C 180,E1 -6566.697,E2 -6566.697} C_VEL
LIN {X 0,Y 487.968,Z 325.747,A -85,B 0,C 180,E1 -6567.524,E2 -6567.524} C_VEL
LIN {X 0,Y 487.856,Z 327.357,A -85,B 0,C 180,E1 -6569.174,E2 -6569.174} C_VEL
LIN {X 0,Y 487.852,Z 327.576,A -85,B 0,C 180,E1 -6570,E2 -6570} C_VEL
LIN {X 0,Y 487.899,Z 326.75,A -85,B 0,C 180,E1 -6571.651,E2 -6571.651} C_VEL
LIN {X 0,Y 487.968,Z 325.751,A -85,B 0,C 180,E1 -6572.476,E2 -6572.476} C_VEL
LIN {X 0,Y 487.997,Z 324.348,A -85,B 0,C 180,E1 -6573.302,E2 -6573.302} C_VEL
LIN {X 0,Y 487.92,Z 321.39,A -85,B 0,C 180,E1 -6574.544,E2 -6574.544} C_VEL
LIN {X 0,Y 487.974,Z 317.398,A -85,B 0,C 180,E1 -6575.786,E2 -6575.786} C_VEL
LIN {X 0,Y 488.113,Z 311.27,A -85,B 0,C 180,E1 -6577.238,E2 -6577.238} C_VEL
LIN {X 0,Y 488.285,Z 304.574,A -85,B 0,C 180,E1 -6578.484,E2 -6578.484} C_VEL
LIN {X 0,Y 488.52,Z 296.279,A -85,B 0,C 180,E1 -6579.732,E2 -6579.732} C_VEL
LIN {X 0,Y 488.925,Z 287.805,A -85,B 0,C 180,E1 -6580.77,E2 -6580.77} C_VEL
LIN {X 0,Y 489.329,Z 277.417,A -85,B 0,C 180,E1 -6581.804,E2 -6581.804} C_VEL
LIN {X 0,Y 489.71,Z 266.238,A -85,B 0,C 180,E1 -6582.7,E2 -6582.7} C_VEL
LIN {X 0,Y 490.176,Z 253.873,A -85,B 0,C 180,E1 -6583.473,E2 -6583.473} C_VEL
LIN {X 0,Y 490.618,Z 241.72,A -85,B 0,C 180,E1 -6584.042,E2 -6584.042} C_VEL
LIN {X 0,Y 490.991,Z 228.487,A -85,B 0,C 180,E1 -6584.48,E2 -6584.48} C_VEL
LIN {X 0,Y 491.207,Z 215.539,A -85,B 0,C 180,E1 -6584.739,E2 -6584.739} C_VEL
LIN {X 0,Y 491.575,Z 130.433,A -85,B 0,C 180,E1 -6585.999,E2 -6585.999} C_VEL
LIN {X 0,Y 489.215,Z 113.733,A -85,B 0,C 180,E1 -6586.359,E2 -6586.359} C_VEL
LIN {X 0,Y 489.847,Z 93.752,A -85,B 0,C 180,E1 -6589.486,E2 -6589.486} C_VEL
LIN {X 0,Y 490.464,Z 74.557,A -85,B 0,C 180,E1 -6592.539,E2 -6592.539} C_VEL
LIN {X 0,Y 490.893,Z 62.228,A -85,B 0,C 180,E1 -6594.531,E2 -6594.531} C_VEL
LIN {X 0,Y 488.814,Z 51.599,A -85,B 0,C 180,E1 -6596.411,E2 -6596.411} C_VEL
LIN {X 0,Y 488.726,Z 51.605,A -85,B 0,C 180,E1 -6599.27,E2 -6599.27} C_VEL
LIN {X 0,Y 488.705,Z 51.613,A -85,B 0,C 180,E1 -6602.147,E2 -6602.147} C_VEL
LIN {X 0,Y 488.718,Z 51.605,A -85,B 0,C 180,E1 -6605.115,E2 -6605.115} C_VEL
LIN {X 0,Y 488.683,Z 51.611,A -85,B 0,C 180,E1 -6608.2,E2 -6608.2} C_VEL
LIN {X 0,Y 488.721,Z 51.606,A -85,B 0,C 180,E1 -6610.345,E2 -6610.345} C_VEL
LIN {X 0,Y 488.688,Z 51.614,A -85,B 0,C 180,E1 -6613.655,E2 -6613.655} C_VEL
LIN {X 0,Y 488.687,Z 51.607,A -85,B 0,C 180,E1 -6616.345,E2 -6616.345} C_VEL
LIN {X 0,Y 488.736,Z 51.604,A -85,B 0,C 180,E1 -6619.677,E2 -6619.677} C_VEL
LIN {X 0,Y 488.683,Z 51.609,A -85,B 0,C 180,E1 -6622.841,E2 -6622.841} C_VEL
LIN {X 0,Y 488.728,Z 51.601,A -85,B 0,C 180,E1 -6625.887,E2 -6625.887} C_VEL
LIN {X 0,Y 488.696,Z 51.612,A -85,B 0,C 180,E1 -6628.82,E2 -6628.82} C_VEL
LIN {X 0,Y 488.749,Z 51.602,A -85,B 0,C 180,E1 -6631.671,E2 -6631.671} C_VEL
LIN {X 0,Y 488.743,Z 51.601,A -85,B 0,C 180,E1 -6634.444,E2 -6634.444} C_VEL
LIN {X 0,Y 488.726,Z 51.604,A -85,B 0,C 180,E1 -6637.153,E2 -6637.153} C_VEL
LIN {X 0,Y 488.728,Z 51.602,A -85,B 0,C 180,E1 -6639.81,E2 -6639.81} C_VEL
LIN {X 0,Y 488.732,Z 51.607,A -85,B 0,C 180,E1 -6642.423,E2 -6642.423} C_VEL
LIN {X 0,Y 488.767,Z 51.6,A -85,B 0,C 180,E1 -6645,E2 -6645} C_VEL
LIN {X 0,Y 488.81,Z 51.596,A -85,B 0,C 180,E1 -6648.388,E2 -6648.388} C_VEL
LIN {X 0,Y 488.821,Z 51.594,A -85,B 0,C 180,E1 -6651.734,E2 -6651.734} C_VEL
LIN {X 0,Y 488.854,Z 51.593,A -85,B 0,C 180,E1 -6654.224,E2 -6654.224} C_VEL
LIN {X 0,Y 488.959,Z 51.576,A -85,B 0,C 180,E1 -6657.529,E2 -6657.529} C_VEL
LIN {X 0,Y 488.939,Z 51.577,A -85,B 0,C 180,E1 -6660.823,E2 -6660.823} C_VEL
LIN {X 0,Y 488.963,Z 51.572,A -85,B 0,C 180,E1 -6662.471,E2 -6662.471} C_VEL
LIN {X 0,Y 488.841,Z 51.595,A -85,B 0,C 180,E1 -6665.776,E2 -6665.776} C_VEL
LIN {X 0,Y 488.789,Z 51.592,A -85,B 0,C 180,E1 -6668.267,E2 -6668.267} C_VEL
LIN {X 0,Y 488.81,Z 51.597,A -85,B 0,C 180,E1 -6671.612,E2 -6671.612} C_VEL
LIN {X 0,Y 488.766,Z 51.6,A -85,B 0,C 180,E1 -6675,E2 -6675} C_VEL
LIN {X 0,Y 488.749,Z 51.599,A -85,B 0,C 180,E1 -6678.442,E2 -6678.442} C_VEL
LIN {X 0,Y 488.711,Z 51.611,A -85,B 0,C 180,E1 -6681.071,E2 -6681.071} C_VEL
LIN {X 0,Y 488.691,Z 51.606,A -85,B 0,C 180,E1 -6683.746,E2 -6683.746} C_VEL
LIN {X 0,Y 488.722,Z 51.608,A -85,B 0,C 180,E1 -6686.474,E2 -6686.474} C_VEL
LIN {X 0,Y 488.713,Z 51.606,A -85,B 0,C 180,E1 -6689.271,E2 -6689.271} C_VEL
LIN {X 0,Y 488.705,Z 51.609,A -85,B 0,C 180,E1 -6692.147,E2 -6692.147} C_VEL
LIN {X 0,Y 488.715,Z 51.606,A -85,B 0,C 180,E1 -6695.115,E2 -6695.115} C_VEL
LIN {X 0,Y 488.678,Z 51.616,A -85,B 0,C 180,E1 -6698.2,E2 -6698.2} C_VEL
LIN {X 0,Y 488.72,Z 51.603,A -85,B 0,C 180,E1 -6700.344,E2 -6700.344} C_VEL
LIN {X 0,Y 488.679,Z 51.614,A -85,B 0,C 180,E1 -6703.655,E2 -6703.655} C_VEL
LIN {X 0,Y 488.678,Z 51.614,A -85,B 0,C 180,E1 -6706.344,E2 -6706.344} C_VEL
LIN {X 0,Y 488.704,Z 51.613,A -85,B 0,C 180,E1 -6709.673,E2 -6709.673} C_VEL
LIN {X 0,Y 488.671,Z 51.612,A -85,B 0,C 180,E1 -6712.84,E2 -6712.84} C_VEL
LIN {X 0,Y 488.725,Z 51.61,A -85,B 0,C 180,E1 -6715.886,E2 -6715.886} C_VEL
LIN {X 0,Y 488.692,Z 51.615,A -85,B 0,C 180,E1 -6718.82,E2 -6718.82} C_VEL
LIN {X 0,Y 488.78,Z 51.702,A -85,B 0,C 180,E1 -6720.805,E2 -6720.805} C_VEL
LIN {X 0,Y 489.657,Z 57.867,A -85,B 0,C 180,E1 -6722.194,E2 -6722.194} C_VEL
LIN {X 0,Y 489.618,Z 60.736,A -85,B 0,C 180,E1 -6722.812,E2 -6722.812} C_VEL
LIN {X 0,Y 489.361,Z 63.119,A -85,B 0,C 180,E1 -6723.16,E2 -6723.16} C_VEL
LIN {X 0,Y 488.666,Z 67.091,A -85,B 0,C 180,E1 -6723.475,E2 -6723.475} C_VEL
LIN {X 0,Y 487.76,Z 71.648,A -85,B 0,C 180,E1 -6723.676,E2 -6723.676} C_VEL
LIN {X 0,Y 486.552,Z 77.696,A -85,B 0,C 180,E1 -6723.805,E2 -6723.805} C_VEL
LIN {X 0,Y 485.328,Z 86.135,A -85,B 0,C 180,E1 -6723.898,E2 -6723.898} C_VEL
LIN {X 0,Y 485.167,Z 90.384,A -85,B 0,C 180,E1 -6723.957,E2 -6723.957} C_VEL
LIN {X 0,Y 484.503,Z 172.434,A -85,B 0,C 180,E1 -6725.209,E2 -6725.209} C_VEL
LIN {X 0,Y 484.321,Z 185.95,A -85,B 0,C 180,E1 -6725.599,E2 -6725.599} C_VEL
LIN {X 0,Y 484.067,Z 197.722,A -85,B 0,C 180,E1 -6726.099,E2 -6726.099} C_VEL
LIN {X 0,Y 483.612,Z 210.087,A -85,B 0,C 180,E1 -6726.807,E2 -6726.807} C_VEL
LIN {X 0,Y 483.125,Z 221.607,A -85,B 0,C 180,E1 -6727.664,E2 -6727.664} C_VEL
LIN {X 0,Y 482.73,Z 232.183,A -85,B 0,C 180,E1 -6728.656,E2 -6728.656} C_VEL
LIN {X 0,Y 482.26,Z 241.563,A -85,B 0,C 180,E1 -6729.75,E2 -6729.75} C_VEL
LIN {X 0,Y 481.82,Z 250.628,A -85,B 0,C 180,E1 -6731.062,E2 -6731.062} C_VEL
LIN {X 0,Y 481.547,Z 257.805,A -85,B 0,C 180,E1 -6732.372,E2 -6732.372} C_VEL
LIN {X 0,Y 481.238,Z 264.291,A -85,B 0,C 180,E1 -6733.89,E2 -6733.89} C_VEL
LIN {X 0,Y 481.101,Z 268.505,A -85,B 0,C 180,E1 -6735.188,E2 -6735.188} C_VEL
LIN {X 0,Y 480.96,Z 271.607,A -85,B 0,C 180,E1 -6736.479,E2 -6736.479} C_VEL
LIN {X 0,Y 480.915,Z 273.127,A -85,B 0,C 180,E1 -6737.338,E2 -6737.338} C_VEL
LIN {X 0,Y 480.886,Z 274.268,A -85,B 0,C 180,E1 -6738.289,E2 -6738.289} C_VEL
LIN {X 0,Y 480.85,Z 275.095,A -85,B 0,C 180,E1 -6739.899,E2 -6739.899} C_VEL
LIN {X 0,Y 480.837,Z 274.95,A -85,B 0,C 180,E1 -6740.748,E2 -6740.748} C_VEL
LIN {X 0,Y 480.887,Z 274.372,A -85,B 0,C 180,E1 -6741.596,E2 -6741.596} C_VEL
LIN {X 0,Y 481.001,Z 272.056,A -85,B 0,C 180,E1 -6743.287,E2 -6743.287} C_VEL
LIN {X 0,Y 481.038,Z 269.207,A -85,B 0,C 180,E1 -6744.551,E2 -6744.551} C_VEL
LIN {X 0,Y 481.188,Z 265.336,A -85,B 0,C 180,E1 -6745.812,E2 -6745.812} C_VEL
LIN {X 0,Y 481.333,Z 260.356,A -85,B 0,C 180,E1 -6747.071,E2 -6747.071} C_VEL
LIN {X 0,Y 481.543,Z 254.109,A -85,B 0,C 180,E1 -6748.327,E2 -6748.327} C_VEL
LIN {X 0,Y 481.897,Z 246.291,A -85,B 0,C 180,E1 -6749.582,E2 -6749.582} C_VEL
LIN {X 0,Y 482.267,Z 236.599,A -85,B 0,C 180,E1 -6750.835,E2 -6750.835} C_VEL
LIN {X 0,Y 482.736,Z 226.479,A -85,B 0,C 180,E1 -6751.877,E2 -6751.877} C_VEL
LIN {X 0,Y 483.179,Z 216.468,A -85,B 0,C 180,E1 -6752.71,E2 -6752.71} C_VEL
LIN {X 0,Y 483.602,Z 205.57,A -85,B 0,C 180,E1 -6753.437,E2 -6753.437} C_VEL
LIN {X 0,Y 483.871,Z 193.562,A -85,B 0,C 180,E1 -6754.06,E2 -6754.06} C_VEL
LIN {X 0,Y 484.095,Z 181.021,A -85,B 0,C 180,E1 -6754.528,E2 -6754.528} C_VEL
LIN {X 0,Y 484.298,Z 167.827,A -85,B 0,C 180,E1 -6754.839,E2 -6754.839} C_VEL
LIN {X 0,Y 484.9,Z 77.275,A -85,B 0,C 180,E1 -6756.188,E2 -6756.188} C_VEL
LIN {X 0,Y 482.452,Z 65.175,A -85,B 0,C 180,E1 -6756.456,E2 -6756.456} C_VEL
LIN {X 0,Y 482.575,Z 58.017,A -85,B 0,C 180,E1 -6757.978,E2 -6757.978} C_VEL
LIN {X 0,Y 481.737,Z 52.481,A -85,B 0,C 180,E1 -6759.235,E2 -6759.235} C_VEL
LIN {X 0,Y 481.755,Z 52.473,A -85,B 0,C 180,E1 -6762.2,E2 -6762.2} C_VEL
LIN {X 0,Y 481.728,Z 52.475,A -85,B 0,C 180,E1 -6765.659,E2 -6765.659} C_VEL
LIN {X 0,Y 481.714,Z 52.48,A -85,B 0,C 180,E1 -6768.722,E2 -6768.722} C_VEL
LIN {X 0,Y 481.647,Z 52.484,A -85,B 0,C 180,E1 -6771.395,E2 -6771.395} C_VEL
LIN {X 0,Y 481.663,Z 52.489,A -85,B 0,C 180,E1 -6774.114,E2 -6774.114} C_VEL
LIN {X 0,Y 481.749,Z 52.472,A -85,B 0,C 180,E1 -6777.139,E2 -6777.139} C_VEL
LIN {X 0,Y 481.681,Z 52.485,A -85,B 0,C 180,E1 -6779.741,E2 -6779.741} C_VEL
LIN {X 0,Y 481.674,Z 52.482,A -85,B 0,C 180,E1 -6782.674,E2 -6782.674} C_VEL
LIN {X 0,Y 481.644,Z 52.492,A -85,B 0,C 180,E1 -6785.709,E2 -6785.709} C_VEL
LIN {X 0,Y 481.673,Z 52.481,A -85,B 0,C 180,E1 -6788.859,E2 -6788.859} C_VEL
LIN {X 0,Y 481.655,Z 52.487,A -85,B 0,C 180,E1 -6791.913,E2 -6791.913} C_VEL
LIN {X 0,Y 481.657,Z 52.483,A -85,B 0,C 180,E1 -6794.458,E2 -6794.458} C_VEL
LIN {X 0,Y 481.65,Z 52.486,A -85,B 0,C 180,E1 -6797.84,E2 -6797.84} C_VEL
LIN {X 0,Y 481.664,Z 52.484,A -85,B 0,C 180,E1 -6800.654,E2 -6800.654} C_VEL
LIN {X 0,Y 481.631,Z 52.492,A -85,B 0,C 180,E1 -6803.376,E2 -6803.376} C_VEL
LIN {X 0,Y 481.713,Z 52.477,A -85,B 0,C 180,E1 -6806.33,E2 -6806.33} C_VEL
LIN {X 0,Y 481.655,Z 52.486,A -85,B 0,C 180,E1 -6809.418,E2 -6809.418} C_VEL
LIN {X 0,Y 481.704,Z 52.478,A -85,B 0,C 180,E1 -6812.168,E2 -6812.168} C_VEL
LIN {X 0,Y 481.72,Z 52.481,A -85,B 0,C 180,E1 -6814.97,E2 -6814.97} C_VEL
LIN {X 0,Y 481.653,Z 52.484,A -85,B 0,C 180,E1 -6817.705,E2 -6817.705} C_VEL
LIN {X 0,Y 481.708,Z 52.483,A -85,B 0,C 180,E1 -6820.393,E2 -6820.393} C_VEL
LIN {X 0,Y 481.681,Z 52.482,A -85,B 0,C 180,E1 -6823.034,E2 -6823.034} C_VEL
LIN {X 0,Y 481.695,Z 52.479,A -85,B 0,C 180,E1 -6825.639,E2 -6825.639} C_VEL
LIN {X 0,Y 481.756,Z 52.478,A -85,B 0,C 180,E1 -6828.215,E2 -6828.215} C_VEL
LIN {X 0,Y 481.745,Z 52.474,A -85,B 0,C 180,E1 -6831.611,E2 -6831.611} C_VEL
LIN {X 0,Y 481.815,Z 52.471,A -85,B 0,C 180,E1 -6834.14,E2 -6834.14} C_VEL
LIN {X 0,Y 481.926,Z 52.452,A -85,B 0,C 180,E1 -6837.493,E2 -6837.493} C_VEL
LIN {X 0,Y 481.891,Z 52.454,A -85,B 0,C 180,E1 -6840.836,E2 -6840.836} C_VEL
LIN {X 0,Y 481.931,Z 52.45,A -85,B 0,C 180,E1 -6842.508,E2 -6842.508} C_VEL
LIN {X 0,Y 481.796,Z 52.471,A -85,B 0,C 180,E1 -6845.861,E2 -6845.861} C_VEL
LIN {X 0,Y 481.745,Z 52.472,A -85,B 0,C 180,E1 -6848.389,E2 -6848.389} C_VEL
LIN {X 0,Y 481.756,Z 52.474,A -85,B 0,C 180,E1 -6851.785,E2 -6851.785} C_VEL
LIN {X 0,Y 481.748,Z 52.479,A -85,B 0,C 180,E1 -6855.224,E2 -6855.224} C_VEL
LIN {X 0,Y 481.713,Z 52.479,A -85,B 0,C 180,E1 -6858.722,E2 -6858.722} C_VEL
LIN {X 0,Y 481.651,Z 52.488,A -85,B 0,C 180,E1 -6861.395,E2 -6861.395} C_VEL
LIN {X 0,Y 481.662,Z 52.483,A -85,B 0,C 180,E1 -6864.114,E2 -6864.114} C_VEL
LIN {X 0,Y 481.701,Z 52.483,A -85,B 0,C 180,E1 -6867.127,E2 -6867.127} C_VEL
LIN {X 0,Y 481.679,Z 52.481,A -85,B 0,C 180,E1 -6869.741,E2 -6869.741} C_VEL
LIN {X 0,Y 481.675,Z 52.489,A -85,B 0,C 180,E1 -6872.674,E2 -6872.674} C_VEL
LIN {X 0,Y 481.639,Z 52.486,A -85,B 0,C 180,E1 -6875.71,E2 -6875.71} C_VEL
LIN {X 0,Y 481.674,Z 52.484,A -85,B 0,C 180,E1 -6878.859,E2 -6878.859} C_VEL
LIN {X 0,Y 481.656,Z 52.486,A -85,B 0,C 180,E1 -6881.913,E2 -6881.913} C_VEL
LIN {X 0,Y 481.659,Z 52.488,A -85,B 0,C 180,E1 -6884.458,E2 -6884.458} C_VEL
LIN {X 0,Y 481.646,Z 52.489,A -85,B 0,C 180,E1 -6887.839,E2 -6887.839} C_VEL
LIN {X 0,Y 481.66,Z 52.484,A -85,B 0,C 180,E1 -6890.654,E2 -6890.654} C_VEL
LIN {X 0,Y 481.625,Z 52.489,A -85,B 0,C 180,E1 -6893.377,E2 -6893.377} C_VEL
LIN {X 0,Y 481.68,Z 52.482,A -85,B 0,C 180,E1 -6896.327,E2 -6896.327} C_VEL
LIN {X 0,Y 481.653,Z 52.488,A -85,B 0,C 180,E1 -6899.418,E2 -6899.418} C_VEL
LIN {X 0,Y 481.703,Z 52.483,A -85,B 0,C 180,E1 -6902.168,E2 -6902.168} C_VEL
LIN {X 0,Y 481.762,Z 52.583,A -85,B 0,C 180,E1 -6903.726,E2 -6903.726} C_VEL
LIN {X 0,Y 483.736,Z 63.147,A -85,B 0,C 180,E1 -6905.539,E2 -6905.539} C_VEL
LIN {X 0,Y 483.116,Z 82.271,A -85,B 0,C 180,E1 -6908.595,E2 -6908.595} C_VEL
LIN {X 0,Y 482.523,Z 102.263,A -85,B 0,C 180,E1 -6911.751,E2 -6911.751} C_VEL
LIN {X 0,Y 482.127,Z 113.703,A -85,B 0,C 180,E1 -6913.541,E2 -6913.541} C_VEL
LIN {X 0,Y 484.664,Z 133.308,A -85,B 0,C 180,E1 -6913.918,E2 -6913.918} C_VEL
LIN {X 0,Y 484.078,Z 222.369,A -85,B 0,C 180,E1 -6915.254,E2 -6915.254} C_VEL
LIN {X 0,Y 483.778,Z 235.747,A -85,B 0,C 180,E1 -6915.621,E2 -6915.621} C_VEL
LIN {X 0,Y 483.342,Z 247.979,A -85,B 0,C 180,E1 -6916.118,E2 -6916.118} C_VEL
LIN {X 0,Y 482.92,Z 259.508,A -85,B 0,C 180,E1 -6916.749,E2 -6916.749} C_VEL
LIN {X 0,Y 482.444,Z 271.101,A -85,B 0,C 180,E1 -6917.573,E2 -6917.573} C_VEL
LIN {X 0,Y 482.053,Z 281.947,A -85,B 0,C 180,E1 -6918.542,E2 -6918.542} C_VEL
LIN {X 0,Y 481.679,Z 290.618,A -85,B 0,C 180,E1 -6919.491,E2 -6919.491} C_VEL
LIN {X 0,Y 481.392,Z 298.61,A -85,B 0,C 180,E1 -6920.547,E2 -6920.547} C_VEL
LIN {X 0,Y 481.149,Z 306.425,A -85,B 0,C 180,E1 -6921.812,E2 -6921.812} C_VEL
LIN {X 0,Y 480.96,Z 313.604,A -85,B 0,C 180,E1 -6923.287,E2 -6923.287} C_VEL
LIN {X 0,Y 480.907,Z 318.388,A -85,B 0,C 180,E1 -6924.549,E2 -6924.549} C_VEL
LIN {X 0,Y 480.848,Z 322.041,A -85,B 0,C 180,E1 -6925.809,E2 -6925.809} C_VEL
LIN {X 0,Y 480.919,Z 323.933,A -85,B 0,C 180,E1 -6926.649,E2 -6926.649} C_VEL
LIN {X 0,Y 480.878,Z 325.348,A -85,B 0,C 180,E1 -6927.487,E2 -6927.487} C_VEL
LIN {X 0,Y 480.831,Z 326.354,A -85,B 0,C 180,E1 -6928.325,E2 -6928.325} C_VEL
LIN {X 0,Y 480.774,Z 327.192,A -85,B 0,C 180,E1 -6930,E2 -6930} C_VEL
LIN {X 0,Y 480.781,Z 326.982,A -85,B 0,C 180,E1 -6930.838,E2 -6930.838} C_VEL
LIN {X 0,Y 480.831,Z 326.376,A -85,B 0,C 180,E1 -6931.675,E2 -6931.675} C_VEL
LIN {X 0,Y 480.878,Z 325.38,A -85,B 0,C 180,E1 -6932.513,E2 -6932.513} C_VEL
LIN {X 0,Y 480.918,Z 323.984,A -85,B 0,C 180,E1 -6933.351,E2 -6933.351} C_VEL
LIN {X 0,Y 480.838,Z 321.034,A -85,B 0,C 180,E1 -6934.611,E2 -6934.611} C_VEL
LIN {X 0,Y 480.876,Z 317.052,A -85,B 0,C 180,E1 -6935.872,E2 -6935.872} C_VEL
LIN {X 0,Y 481.033,Z 310.945,A -85,B 0,C 180,E1 -6937.345,E2 -6937.345} C_VEL
LIN {X 0,Y 481.227,Z 304.268,A -85,B 0,C 180,E1 -6938.609,E2 -6938.609} C_VEL
LIN {X 0,Y 481.478,Z 295.996,A -85,B 0,C 180,E1 -6939.876,E2 -6939.876} C_VEL
LIN {X 0,Y 481.927,Z 287.553,A -85,B 0,C 180,E1 -6940.928,E2 -6940.928} C_VEL
LIN {X 0,Y 482.333,Z 277.415,A -85,B 0,C 180,E1 -6941.959,E2 -6941.959} C_VEL
LIN {X 0,Y 482.711,Z 267.155,A -85,B 0,C 180,E1 -6942.807,E2 -6942.807} C_VEL
LIN {X 0,Y 483.205,Z 255.647,A -85,B 0,C 180,E1 -6943.564,E2 -6943.564} C_VEL
LIN {X 0,Y 483.677,Z 243.086,A -85,B 0,C 180,E1 -6944.194,E2 -6944.194} C_VEL
LIN {X 0,Y 484.113,Z 229.664,A -85,B 0,C 180,E1 -6944.664,E2 -6944.664} C_VEL
LIN {X 0,Y 484.373,Z 216.432,A -85,B 0,C 180,E1 -6944.951,E2 -6944.951} C_VEL
LIN {X 0,Y 484.851,Z 131.609,A -85,B 0,C 180,E1 -6946.224,E2 -6946.224} C_VEL
LIN {X 0,Y 482.241,Z 113.371,A -85,B 0,C 180,E1 -6946.619,E2 -6946.619} C_VEL
LIN {X 0,Y 482.899,Z 93.527,A -85,B 0,C 180,E1 -6949.778,E2 -6949.778} C_VEL
LIN {X 0,Y 483.544,Z 75.737,A -85,B 0,C 180,E1 -6952.654,E2 -6952.654} C_VEL
LIN {X 0,Y 484.059,Z 64.799,A -85,B 0,C 180,E1 -6954.443,E2 -6954.443} C_VEL
LIN {X 0,Y 482.337,Z 55.19,A -85,B 0,C 180,E1 -6956.153,E2 -6956.153} C_VEL
LIN {X 0,Y 481.774,Z 52.477,A -85,B 0,C 180,E1 -6956.652,E2 -6956.652} C_VEL
LIN {X 0,Y 481.682,Z 52.484,A -85,B 0,C 180,E1 -6959.741,E2 -6959.741} C_VEL
LIN {X 0,Y 481.673,Z 52.486,A -85,B 0,C 180,E1 -6962.674,E2 -6962.674} C_VEL
LIN {X 0,Y 481.639,Z 52.491,A -85,B 0,C 180,E1 -6965.71,E2 -6965.71} C_VEL
LIN {X 0,Y 481.674,Z 52.479,A -85,B 0,C 180,E1 -6968.859,E2 -6968.859} C_VEL
LIN {X 0,Y 481.656,Z 52.488,A -85,B 0,C 180,E1 -6971.913,E2 -6971.913} C_VEL
LIN {X 0,Y 481.658,Z 52.482,A -85,B 0,C 180,E1 -6974.458,E2 -6974.458} C_VEL
LIN {X 0,Y 481.651,Z 52.487,A -85,B 0,C 180,E1 -6977.839,E2 -6977.839} C_VEL
LIN {X 0,Y 481.664,Z 52.48,A -85,B 0,C 180,E1 -6980.654,E2 -6980.654} C_VEL
LIN {X 0,Y 481.631,Z 52.49,A -85,B 0,C 180,E1 -6983.376,E2 -6983.376} C_VEL
LIN {X 0,Y 481.68,Z 52.478,A -85,B 0,C 180,E1 -6986.327,E2 -6986.327} C_VEL
LIN {X 0,Y 481.655,Z 52.485,A -85,B 0,C 180,E1 -6989.417,E2 -6989.417} C_VEL
LIN {X 0,Y 481.704,Z 52.479,A -85,B 0,C 180,E1 -6992.168,E2 -6992.168} C_VEL
LIN {X 0,Y 481.715,Z 52.482,A -85,B 0,C 180,E1 -6994.97,E2 -6994.97} C_VEL
LIN {X 0,Y 481.653,Z 52.482,A -85,B 0,C 180,E1 -6997.705,E2 -6997.705} C_VEL
LIN {X 0,Y 481.708,Z 52.482,A -85,B 0,C 180,E1 -7000.393,E2 -7000.393} C_VEL
LIN {X 0,Y 481.692,Z 52.478,A -85,B 0,C 180,E1 -7003.034,E2 -7003.034} C_VEL
LIN {X 0,Y 481.694,Z 52.48,A -85,B 0,C 180,E1 -7005.639,E2 -7005.639} C_VEL
LIN {X 0,Y 481.756,Z 52.473,A -85,B 0,C 180,E1 -7008.215,E2 -7008.215} C_VEL
LIN {X 0,Y 481.766,Z 52.472,A -85,B 0,C 180,E1 -7011.612,E2 -7011.612} C_VEL
LIN {X 0,Y 481.815,Z 52.468,A -85,B 0,C 180,E1 -7014.139,E2 -7014.139} C_VEL
LIN {X 0,Y 481.925,Z 52.452,A -85,B 0,C 180,E1 -7017.492,E2 -7017.492} C_VEL
LIN {X 0,Y 481.89,Z 52.455,A -85,B 0,C 180,E1 -7020.836,E2 -7020.836} C_VEL
LIN {X 0,Y 481.93,Z 52.448,A -85,B 0,C 180,E1 -7022.507,E2 -7022.507} C_VEL
LIN {X 0,Y 481.802,Z 52.47,A -85,B 0,C 180,E1 -7025.86,E2 -7025.86} C_VEL
LIN {X 0,Y 481.744,Z 52.469,A -85,B 0,C 180,E1 -7028.389,E2 -7028.389} C_VEL
LIN {X 0,Y 481.755,Z 52.474,A -85,B 0,C 180,E1 -7031.785,E2 -7031.785} C_VEL
LIN {X 0,Y 481.747,Z 52.478,A -85,B 0,C 180,E1 -7035.224,E2 -7035.224} C_VEL
LIN {X 0,Y 481.711,Z 52.478,A -85,B 0,C 180,E1 -7038.722,E2 -7038.722} C_VEL
LIN {X 0,Y 481.649,Z 52.487,A -85,B 0,C 180,E1 -7041.394,E2 -7041.394} C_VEL
LIN {X 0,Y 481.674,Z 52.481,A -85,B 0,C 180,E1 -7044.113,E2 -7044.113} C_VEL
LIN {X 0,Y 481.697,Z 52.48,A -85,B 0,C 180,E1 -7047.127,E2 -7047.127} C_VEL
LIN {X 0,Y 481.676,Z 52.482,A -85,B 0,C 180,E1 -7049.741,E2 -7049.741} C_VEL
LIN {X 0,Y 481.673,Z 52.487,A -85,B 0,C 180,E1 -7052.674,E2 -7052.674} C_VEL
LIN {X 0,Y 481.633,Z 52.488,A -85,B 0,C 180,E1 -7055.71,E2 -7055.71} C_VEL
LIN {X 0,Y 481.671,Z 52.484,A -85,B 0,C 180,E1 -7058.859,E2 -7058.859} C_VEL
LIN {X 0,Y 481.647,Z 52.485,A -85,B 0,C 180,E1 -7061.912,E2 -7061.912} C_VEL
LIN {X 0,Y 481.656,Z 52.488,A -85,B 0,C 180,E1 -7064.458,E2 -7064.458} C_VEL
LIN {X 0,Y 481.644,Z 52.492,A -85,B 0,C 180,E1 -7067.839,E2 -7067.839} C_VEL
LIN {X 0,Y 481.657,Z 52.485,A -85,B 0,C 180,E1 -7070.655,E2 -7070.655} C_VEL
LIN {X 0,Y 481.623,Z 52.495,A -85,B 0,C 180,E1 -7073.377,E2 -7073.377} C_VEL
LIN {X 0,Y 481.678,Z 52.486,A -85,B 0,C 180,E1 -7076.327,E2 -7076.327} C_VEL
LIN {X 0,Y 481.65,Z 52.494,A -85,B 0,C 180,E1 -7079.418,E2 -7079.418} C_VEL
LIN {X 0,Y 481.744,Z 52.682,A -85,B 0,C 180,E1 -7080.634,E2 -7080.634} C_VEL
LIN {X 0,Y 482.726,Z 59.7,A -85,B 0,C 180,E1 -7082.232,E2 -7082.232} C_VEL
LIN {X 0,Y 482.632,Z 65.529,A -85,B 0,C 180,E1 -7083.475,E2 -7083.475} C_VEL
LIN {X 0,Y 485.268,Z 77.772,A -85,B 0,C 180,E1 -7083.768,E2 -7083.768} C_VEL
LIN {X 0,Y 485.167,Z 90.384,A -85,B 0,C 180,E1 -7083.957,E2 -7083.957} C_VEL
LIN {X 0,Y 484.494,Z 96.229,A -85,B 0,C 180,E1 -7084.02,E2 -7084.02} C_VEL
LIN {X 0,Y 478.881,Z 115.249,A -85,B 0,C 180,E1 -7084.096,E2 -7084.096} C_VEL
LIN {X 0,Y 478.166,Z 121.096,A -85,B 0,C 180,E1 -7084.159,E2 -7084.159} C_VEL
LIN {X 0,Y 477.731,Z 172.007,A -85,B 0,C 180,E1 -7084.95,E2 -7084.95} C_VEL
LIN {X 0,Y 477.558,Z 185.003,A -85,B 0,C 180,E1 -7085.318,E2 -7085.318} C_VEL
LIN {X 0,Y 477.248,Z 198.118,A -85,B 0,C 180,E1 -7085.872,E2 -7085.872} C_VEL
LIN {X 0,Y 476.764,Z 209.853,A -85,B 0,C 180,E1 -7086.546,E2 -7086.546} C_VEL
LIN {X 0,Y 476.244,Z 221.747,A -85,B 0,C 180,E1 -7087.438,E2 -7087.438} C_VEL
LIN {X 0,Y 475.838,Z 231.277,A -85,B 0,C 180,E1 -7088.331,E2 -7088.331} C_VEL
LIN {X 0,Y 475.393,Z 240.954,A -85,B 0,C 180,E1 -7089.445,E2 -7089.445} C_VEL
LIN {X 0,Y 474.902,Z 250.185,A -85,B 0,C 180,E1 -7090.775,E2 -7090.775} C_VEL
LIN {X 0,Y 474.552,Z 257.557,A -85,B 0,C 180,E1 -7092.103,E2 -7092.103} C_VEL
LIN {X 0,Y 474.293,Z 262.479,A -85,B 0,C 180,E1 -7093.205,E2 -7093.205} C_VEL
LIN {X 0,Y 474.137,Z 267.215,A -85,B 0,C 180,E1 -7094.525,E2 -7094.525} C_VEL
LIN {X 0,Y 473.969,Z 270.785,A -85,B 0,C 180,E1 -7095.838,E2 -7095.838} C_VEL
LIN {X 0,Y 473.851,Z 273.301,A -85,B 0,C 180,E1 -7097.146,E2 -7097.146} C_VEL
LIN {X 0,Y 473.82,Z 274.634,A -85,B 0,C 180,E1 -7098.224,E2 -7098.224} C_VEL
LIN {X 0,Y 473.759,Z 275.456,A -85,B 0,C 180,E1 -7099.746,E2 -7099.746} C_VEL
LIN {X 0,Y 473.744,Z 275.381,A -85,B 0,C 180,E1 -7100.608,E2 -7100.608} C_VEL
LIN {X 0,Y 473.792,Z 274.88,A -85,B 0,C 180,E1 -7101.47,E2 -7101.47} C_VEL
LIN {X 0,Y 473.902,Z 272.661,A -85,B 0,C 180,E1 -7103.186,E2 -7103.186} C_VEL
LIN {X 0,Y 473.975,Z 269.909,A -85,B 0,C 180,E1 -7104.469,E2 -7104.469} C_VEL
LIN {X 0,Y 474.118,Z 266.146,A -85,B 0,C 180,E1 -7105.75,E2 -7105.75} C_VEL
LIN {X 0,Y 474.248,Z 261.282,A -85,B 0,C 180,E1 -7107.027,E2 -7107.027} C_VEL
LIN {X 0,Y 474.47,Z 255.168,A -85,B 0,C 180,E1 -7108.302,E2 -7108.302} C_VEL
LIN {X 0,Y 474.842,Z 247.554,A -85,B 0,C 180,E1 -7109.576,E2 -7109.576} C_VEL
LIN {X 0,Y 475.23,Z 238.03,A -85,B 0,C 180,E1 -7110.847,E2 -7110.847} C_VEL
LIN {X 0,Y 475.718,Z 228.201,A -85,B 0,C 180,E1 -7111.905,E2 -7111.905} C_VEL
LIN {X 0,Y 476.14,Z 218.521,A -85,B 0,C 180,E1 -7112.75,E2 -7112.75} C_VEL
LIN {X 0,Y 476.599,Z 208.017,A -85,B 0,C 180,E1 -7113.487,E2 -7113.487} C_VEL
LIN {X 0,Y 476.929,Z 195.46,A -85,B 0,C 180,E1 -7114.173,E2 -7114.173} C_VEL
LIN {X 0,Y 477.158,Z 182.893,A -85,B 0,C 180,E1 -7114.673,E2 -7114.673} C_VEL
LIN {X 0,Y 477.384,Z 170.76,A -85,B 0,C 180,E1 -7114.988,E2 -7114.988} C_VEL
LIN {X 0,Y 477.894,Z 77.455,A -85,B 0,C 180,E1 -7116.41,E2 -7116.41} C_VEL
LIN {X 0,Y 475.526,Z 65.476,A -85,B 0,C 180,E1 -7116.684,E2 -7116.684} C_VEL
LIN {X 0,Y 475.577,Z 59.07,A -85,B 0,C 180,E1 -7118.063,E2 -7118.063} C_VEL
LIN {X 0,Y 474.704,Z 53.357,A -85,B 0,C 180,E1 -7119.373,E2 -7119.373} C_VEL
LIN {X 0,Y 474.703,Z 53.353,A -85,B 0,C 180,E1 -7122.276,E2 -7122.276} C_VEL
LIN {X 0,Y 474.683,Z 53.352,A -85,B 0,C 180,E1 -7125.768,E2 -7125.768} C_VEL
LIN {X 0,Y 474.667,Z 53.355,A -85,B 0,C 180,E1 -7129.01,E2 -7129.01} C_VEL
LIN {X 0,Y 474.59,Z 53.365,A -85,B 0,C 180,E1 -7131.729,E2 -7131.729} C_VEL
LIN {X 0,Y 474.643,Z 53.361,A -85,B 0,C 180,E1 -7134.494,E2 -7134.494} C_VEL
LIN {X 0,Y 474.701,Z 53.35,A -85,B 0,C 180,E1 -7137.339,E2 -7137.339} C_VEL
LIN {X 0,Y 474.606,Z 53.362,A -85,B 0,C 180,E1 -7140.81,E2 -7140.81} C_VEL
LIN {X 0,Y 474.641,Z 53.364,A -85,B 0,C 180,E1 -7143.984,E2 -7143.984} C_VEL
LIN {X 0,Y 474.576,Z 53.365,A -85,B 0,C 180,E1 -7146.9,E2 -7146.9} C_VEL
LIN {X 0,Y 474.63,Z 53.367,A -85,B 0,C 180,E1 -7149.648,E2 -7149.648} C_VEL
LIN {X 0,Y 474.617,Z 53.361,A -85,B 0,C 180,E1 -7152.935,E2 -7152.935} C_VEL
LIN {X 0,Y 474.609,Z 53.364,A -85,B 0,C 180,E1 -7155.895,E2 -7155.895} C_VEL
LIN {X 0,Y 474.63,Z 53.363,A -85,B 0,C 180,E1 -7159.041,E2 -7159.041} C_VEL
LIN {X 0,Y 474.613,Z 53.363,A -85,B 0,C 180,E1 -7161.704,E2 -7161.704} C_VEL
LIN {X 0,Y 474.629,Z 53.362,A -85,B 0,C 180,E1 -7164.726,E2 -7164.726} C_VEL
LIN {X 0,Y 474.639,Z 53.358,A -85,B 0,C 180,E1 -7167.788,E2 -7167.788} C_VEL
LIN {X 0,Y 474.629,Z 53.367,A -85,B 0,C 180,E1 -7170.885,E2 -7170.885} C_VEL
LIN {X 0,Y 474.664,Z 53.355,A -85,B 0,C 180,E1 -7173.629,E2 -7173.629} C_VEL
LIN {X 0,Y 474.64,Z 53.365,A -85,B 0,C 180,E1 -7176.642,E2 -7176.642} C_VEL
LIN {X 0,Y 474.658,Z 53.357,A -85,B 0,C 180,E1 -7180.09,E2 -7180.09} C_VEL
LIN {X 0,Y 474.641,Z 53.361,A -85,B 0,C 180,E1 -7182.774,E2 -7182.774} C_VEL
LIN {X 0,Y 474.653,Z 53.356,A -85,B 0,C 180,E1 -7185.421,E2 -7185.421} C_VEL
LIN {X 0,Y 474.71,Z 53.353,A -85,B 0,C 180,E1 -7188.038,E2 -7188.038} C_VEL
LIN {X 0,Y 474.717,Z 53.349,A -85,B 0,C 180,E1 -7191.486,E2 -7191.486} C_VEL
LIN {X 0,Y 474.778,Z 53.348,A -85,B 0,C 180,E1 -7194.052,E2 -7194.052} C_VEL
LIN {X 0,Y 474.892,Z 53.328,A -85,B 0,C 180,E1 -7197.455,E2 -7197.455} C_VEL
LIN {X 0,Y 474.917,Z 53.329,A -85,B 0,C 180,E1 -7200,E2 -7200} C_VEL
LIN {X 0,Y 474.898,Z 53.326,A -85,B 0,C 180,E1 -7202.545,E2 -7202.545} C_VEL
LIN {X 0,Y 474.757,Z 53.347,A -85,B 0,C 180,E1 -7205.948,E2 -7205.948} C_VEL
LIN {X 0,Y 474.717,Z 53.348,A -85,B 0,C 180,E1 -7208.514,E2 -7208.514} C_VEL
LIN {X 0,Y 474.71,Z 53.35,A -85,B 0,C 180,E1 -7211.962,E2 -7211.962} C_VEL
LIN {X 0,Y 474.705,Z 53.355,A -85,B 0,C 180,E1 -7215.456,E2 -7215.456} C_VEL
LIN {X 0,Y 474.667,Z 53.36,A -85,B 0,C 180,E1 -7219.01,E2 -7219.01} C_VEL
LIN {X 0,Y 474.593,Z 53.364,A -85,B 0,C 180,E1 -7221.729,E2 -7221.729} C_VEL
LIN {X 0,Y 474.642,Z 53.359,A -85,B 0,C 180,E1 -7224.494,E2 -7224.494} C_VEL
LIN {X 0,Y 474.641,Z 53.36,A -85,B 0,C 180,E1 -7227.324,E2 -7227.324} C_VEL
LIN {X 0,Y 474.608,Z 53.363,A -85,B 0,C 180,E1 -7230.23,E2 -7230.23} C_VEL
LIN {X 0,Y 474.629,Z 53.36,A -85,B 0,C 180,E1 -7233.221,E2 -7233.221} C_VEL
LIN {X 0,Y 474.592,Z 53.368,A -85,B 0,C 180,E1 -7236.323,E2 -7236.323} C_VEL
LIN {X 0,Y 474.622,Z 53.36,A -85,B 0,C 180,E1 -7239.646,E2 -7239.646} C_VEL
LIN {X 0,Y 474.628,Z 53.366,A -85,B 0,C 180,E1 -7242.237,E2 -7242.237} C_VEL
LIN {X 0,Y 474.62,Z 53.36,A -85,B 0,C 180,E1 -7245.298,E2 -7245.298} C_VEL
LIN {X 0,Y 474.618,Z 53.367,A -85,B 0,C 180,E1 -7248.214,E2 -7248.214} C_VEL
LIN {X 0,Y 474.612,Z 53.363,A -85,B 0,C 180,E1 -7251.542,E2 -7251.542} C_VEL
LIN {X 0,Y 474.624,Z 53.36,A -85,B 0,C 180,E1 -7254.725,E2 -7254.725} C_VEL
LIN {X 0,Y 474.638,Z 53.366,A -85,B 0,C 180,E1 -7257.788,E2 -7257.788} C_VEL
LIN {X 0,Y 474.626,Z 53.363,A -85,B 0,C 180,E1 -7260.885,E2 -7260.885} C_VEL
LIN {X 0,Y 474.709,Z 53.404,A -85,B 0,C 180,E1 -7263.542,E2 -7263.542} C_VEL
LIN {X 0,Y 476.735,Z 63.986,A -85,B 0,C 180,E1 -7265.388,E2 -7265.388} C_VEL
LIN {X 0,Y 476.401,Z 75.213,A -85,B 0,C 180,E1 -7267.216,E2 -7267.216} C_VEL
LIN {X 0,Y 475.699,Z 96.159,A -85,B 0,C 180,E1 -7270.584,E2 -7270.584} C_VEL
LIN {X 0,Y 475.15,Z 113.301,A -85,B 0,C 180,E1 -7273.313,E2 -7273.313} C_VEL
LIN {X 0,Y 477.79,Z 133.425,A -85,B 0,C 180,E1 -7273.71,E2 -7273.71} C_VEL
LIN {X 0,Y 477.16,Z 222.216,A -85,B 0,C 180,E1 -7275.063,E2 -7275.063} C_VEL
LIN {X 0,Y 476.828,Z 235.519,A -85,B 0,C 180,E1 -7275.434,E2 -7275.434} C_VEL
LIN {X 0,Y 476.383,Z 248.288,A -85,B 0,C 180,E1 -7275.966,E2 -7275.966} C_VEL
LIN {X 0,Y 475.925,Z 260.433,A -85,B 0,C 180,E1 -7276.659,E2 -7276.659} C_VEL
LIN {X 0,Y 475.413,Z 271.627,A -85,B 0,C 180,E1 -7277.482,E2 -7277.482} C_VEL
LIN {X 0,Y 475.005,Z 282.446,A -85,B 0,C 180,E1 -7278.478,E2 -7278.478} C_VEL
LIN {X 0,Y 474.573,Z 291.81,A -85,B 0,C 180,E1 -7279.548,E2 -7279.548} C_VEL
LIN {X 0,Y 474.219,Z 300.89,A -85,B 0,C 180,E1 -7280.833,E2 -7280.833} C_VEL
LIN {X 0,Y 474.006,Z 308.206,A -85,B 0,C 180,E1 -7282.117,E2 -7282.117} C_VEL
LIN {X 0,Y 473.892,Z 313.148,A -85,B 0,C 180,E1 -7283.186,E2 -7283.186} C_VEL
LIN {X 0,Y 473.817,Z 317.949,A -85,B 0,C 180,E1 -7284.467,E2 -7284.467} C_VEL
LIN {X 0,Y 473.75,Z 321.617,A -85,B 0,C 180,E1 -7285.746,E2 -7285.746} C_VEL
LIN {X 0,Y 473.841,Z 323.519,A -85,B 0,C 180,E1 -7286.599,E2 -7286.599} C_VEL
LIN {X 0,Y 473.793,Z 324.944,A -85,B 0,C 180,E1 -7287.449,E2 -7287.449} C_VEL
LIN {X 0,Y 473.764,Z 325.957,A -85,B 0,C 180,E1 -7288.3,E2 -7288.3} C_VEL
LIN {X 0,Y 473.698,Z 326.807,A -85,B 0,C 180,E1 -7290,E2 -7290} C_VEL
LIN {X 0,Y 473.708,Z 326.607,A -85,B 0,C 180,E1 -7290.85,E2 -7290.85} C_VEL
LIN {X 0,Y 473.764,Z 326.007,A -85,B 0,C 180,E1 -7291.7,E2 -7291.7} C_VEL
LIN {X 0,Y 473.841,Z 323.626,A -85,B 0,C 180,E1 -7293.401,E2 -7293.401} C_VEL
LIN {X 0,Y 473.76,Z 320.688,A -85,B 0,C 180,E1 -7294.68,E2 -7294.68} C_VEL
LIN {X 0,Y 473.788,Z 316.72,A -85,B 0,C 180,E1 -7295.96,E2 -7295.96} C_VEL
LIN {X 0,Y 473.971,Z 310.639,A -85,B 0,C 180,E1 -7297.455,E2 -7297.455} C_VEL
LIN {X 0,Y 474.137,Z 303.982,A -85,B 0,C 180,E1 -7298.739,E2 -7298.739} C_VEL
LIN {X 0,Y 474.425,Z 295.737,A -85,B 0,C 180,E1 -7300.024,E2 -7300.024} C_VEL
LIN {X 0,Y 474.922,Z 287.327,A -85,B 0,C 180,E1 -7301.092,E2 -7301.092} C_VEL
LIN {X 0,Y 475.344,Z 277.441,A -85,B 0,C 180,E1 -7302.12,E2 -7302.12} C_VEL
LIN {X 0,Y 475.786,Z 266.756,A -85,B 0,C 180,E1 -7303.018,E2 -7303.018} C_VEL
LIN {X 0,Y 476.299,Z 255.612,A -85,B 0,C 180,E1 -7303.765,E2 -7303.765} C_VEL
LIN {X 0,Y 476.82,Z 243.22,A -85,B 0,C 180,E1 -7304.402,E2 -7304.402} C_VEL
LIN {X 0,Y 477.282,Z 230.034,A -85,B 0,C 180,E1 -7304.878,E2 -7304.878} C_VEL
LIN {X 0,Y 477.549,Z 217.317,A -85,B 0,C 180,E1 -7305.17,E2 -7305.17} C_VEL
LIN {X 0,Y 478.141,Z 132.791,A -85,B 0,C 180,E1 -7306.458,E2 -7306.458} C_VEL
LIN {X 0,Y 475.27,Z 113,A -85,B 0,C 180,E1 -7306.893,E2 -7306.893} C_VEL
LIN {X 0,Y 475.921,Z 94.691,A -85,B 0,C 180,E1 -7309.855,E2 -7309.855} C_VEL
LIN {X 0,Y 476.623,Z 76.928,A -85,B 0,C 180,E1 -7312.772,E2 -7312.772} C_VEL
LIN {X 0,Y 477.151,Z 66.006,A -85,B 0,C 180,E1 -7314.589,E2 -7314.589} C_VEL
LIN {X 0,Y 475.394,Z 56.416,A -85,B 0,C 180,E1 -7316.328,E2 -7316.328} C_VEL
LIN {X 0,Y 474.707,Z 53.356,A -85,B 0,C 180,E1 -7316.903,E2 -7316.903} C_VEL
LIN {X 0,Y 474.608,Z 53.367,A -85,B 0,C 180,E1 -7320.23,E2 -7320.23} C_VEL
LIN {X 0,Y 474.628,Z 53.362,A -85,B 0,C 180,E1 -7323.221,E2 -7323.221} C_VEL
LIN {X 0,Y 474.592,Z 53.368,A -85,B 0,C 180,E1 -7326.324,E2 -7326.324} C_VEL
LIN {X 0,Y 474.63,Z 53.358,A -85,B 0,C 180,E1 -7329.648,E2 -7329.648} C_VEL
LIN {X 0,Y 474.618,Z 53.36,A -85,B 0,C 180,E1 -7332.934,E2 -7332.934} C_VEL
LIN {X 0,Y 474.609,Z 53.364,A -85,B 0,C 180,E1 -7335.895,E2 -7335.895} C_VEL
LIN {X 0,Y 474.631,Z 53.36,A -85,B 0,C 180,E1 -7339.041,E2 -7339.041} C_VEL
LIN {X 0,Y 474.613,Z 53.363,A -85,B 0,C 180,E1 -7341.704,E2 -7341.704} C_VEL
LIN {X 0,Y 474.626,Z 53.36,A -85,B 0,C 180,E1 -7344.726,E2 -7344.726} C_VEL
LIN {X 0,Y 474.638,Z 53.359,A -85,B 0,C 180,E1 -7347.788,E2 -7347.788} C_VEL
LIN {X 0,Y 474.628,Z 53.362,A -85,B 0,C 180,E1 -7350.884,E2 -7350.884} C_VEL
LIN {X 0,Y 474.662,Z 53.353,A -85,B 0,C 180,E1 -7353.628,E2 -7353.628} C_VEL
LIN {X 0,Y 474.639,Z 53.364,A -85,B 0,C 180,E1 -7356.641,E2 -7356.641} C_VEL
LIN {X 0,Y 474.658,Z 53.357,A -85,B 0,C 180,E1 -7360.09,E2 -7360.09} C_VEL
LIN {X 0,Y 474.651,Z 53.357,A -85,B 0,C 180,E1 -7362.774,E2 -7362.774} C_VEL
LIN {X 0,Y 474.652,Z 53.357,A -85,B 0,C 180,E1 -7365.421,E2 -7365.421} C_VEL
LIN {X 0,Y 474.709,Z 53.35,A -85,B 0,C 180,E1 -7368.038,E2 -7368.038} C_VEL
LIN {X 0,Y 474.731,Z 53.347,A -85,B 0,C 180,E1 -7371.486,E2 -7371.486} C_VEL
LIN {X 0,Y 474.777,Z 53.343,A -85,B 0,C 180,E1 -7374.052,E2 -7374.052} C_VEL
LIN {X 0,Y 474.891,Z 53.328,A -85,B 0,C 180,E1 -7377.455,E2 -7377.455} C_VEL
LIN {X 0,Y 474.916,Z 53.329,A -85,B 0,C 180,E1 -7380,E2 -7380} C_VEL
LIN {X 0,Y 474.896,Z 53.324,A -85,B 0,C 180,E1 -7382.545,E2 -7382.545} C_VEL
LIN {X 0,Y 474.765,Z 53.346,A -85,B 0,C 180,E1 -7385.948,E2 -7385.948} C_VEL
LIN {X 0,Y 474.715,Z 53.345,A -85,B 0,C 180,E1 -7388.514,E2 -7388.514} C_VEL
LIN {X 0,Y 474.708,Z 53.35,A -85,B 0,C 180,E1 -7391.962,E2 -7391.962} C_VEL
LIN {X 0,Y 474.704,Z 53.355,A -85,B 0,C 180,E1 -7395.455,E2 -7395.455} C_VEL
LIN {X 0,Y 474.665,Z 53.357,A -85,B 0,C 180,E1 -7399.01,E2 -7399.01} C_VEL
LIN {X 0,Y 474.592,Z 53.364,A -85,B 0,C 180,E1 -7401.729,E2 -7401.729} C_VEL
LIN {X 0,Y 474.653,Z 53.359,A -85,B 0,C 180,E1 -7404.493,E2 -7404.493} C_VEL
LIN {X 0,Y 474.639,Z 53.358,A -85,B 0,C 180,E1 -7407.324,E2 -7407.324} C_VEL
LIN {X 0,Y 474.606,Z 53.366,A -85,B 0,C 180,E1 -7410.23,E2 -7410.23} C_VEL
LIN {X 0,Y 474.627,Z 53.359,A -85,B 0,C 180,E1 -7413.221,E2 -7413.221} C_VEL
LIN {X 0,Y 474.586,Z 53.371,A -85,B 0,C 180,E1 -7416.324,E2 -7416.324} C_VEL
LIN {X 0,Y 474.626,Z 53.361,A -85,B 0,C 180,E1 -7419.548,E2 -7419.548} C_VEL
LIN {X 0,Y 474.601,Z 53.368,A -85,B 0,C 180,E1 -7422.233,E2 -7422.233} C_VEL
LIN {X 0,Y 474.618,Z 53.363,A -85,B 0,C 180,E1 -7425.298,E2 -7425.298} C_VEL
LIN {X 0,Y 474.616,Z 53.366,A -85,B 0,C 180,E1 -7428.214,E2 -7428.214} C_VEL
LIN {X 0,Y 474.609,Z 53.368,A -85,B 0,C 180,E1 -7431.542,E2 -7431.542} C_VEL
LIN {X 0,Y 474.621,Z 53.364,A -85,B 0,C 180,E1 -7434.725,E2 -7434.725} C_VEL
LIN {X 0,Y 474.636,Z 53.367,A -85,B 0,C 180,E1 -7437.788,E2 -7437.788} C_VEL
LIN {X 0,Y 474.643,Z 53.368,A -85,B 0,C 180,E1 -7440.384,E2 -7440.384} C_VEL
LIN {X 0,Y 475.679,Z 59.387,A -85,B 0,C 180,E1 -7441.784,E2 -7441.784} C_VEL
LIN {X 0,Y 475.71,Z 65.999,A -85,B 0,C 180,E1 -7443.2,E2 -7443.2} C_VEL
LIN {X 0,Y 478.541,Z 78.711,A -85,B 0,C 180,E1 -7443.515,E2 -7443.515} C_VEL
LIN {X 0,Y 478.166,Z 121.096,A -85,B 0,C 180,E1 -7444.159,E2 -7444.159} C_VEL
LIN {X 0,Y 477.443,Z 126.942,A -85,B 0,C 180,E1 -7444.222,E2 -7444.222} C_VEL
LIN {X 0,Y 471.788,Z 145.95,A -85,B 0,C 180,E1 -7444.298,E2 -7444.298} C_VEL
LIN {X 0,Y 471.132,Z 151.793,A -85,B 0,C 180,E1 -7444.364,E2 -7444.364} C_VEL
LIN {X 0,Y 470.918,Z 174.063,A -85,B 0,C 180,E1 -7444.739,E2 -7444.739} C_VEL
LIN {X 0,Y 470.703,Z 187.28,A -85,B 0,C 180,E1 -7445.14,E2 -7445.14} C_VEL
LIN {X 0,Y 470.376,Z 199.813,A -85,B 0,C 180,E1 -7445.702,E2 -7445.702} C_VEL
LIN {X 0,Y 469.881,Z 211.625,A -85,B 0,C 180,E1 -7446.415,E2 -7446.415} C_VEL
LIN {X 0,Y 469.327,Z 223.255,A -85,B 0,C 180,E1 -7447.319,E2 -7447.319} C_VEL
LIN {X 0,Y 468.88,Z 233.505,A -85,B 0,C 180,E1 -7448.328,E2 -7448.328} C_VEL
LIN {X 0,Y 468.405,Z 242.035,A -85,B 0,C 180,E1 -7449.354,E2 -7449.354} C_VEL
LIN {X 0,Y 467.906,Z 251.146,A -85,B 0,C 180,E1 -7450.704,E2 -7450.704} C_VEL
LIN {X 0,Y 467.513,Z 258.382,A -85,B 0,C 180,E1 -7452.051,E2 -7452.051} C_VEL
LIN {X 0,Y 467.216,Z 264.084,A -85,B 0,C 180,E1 -7453.393,E2 -7453.393} C_VEL
LIN {X 0,Y 467.016,Z 268.622,A -85,B 0,C 180,E1 -7454.766,E2 -7454.766} C_VEL
LIN {X 0,Y 466.845,Z 271.838,A -85,B 0,C 180,E1 -7456.062,E2 -7456.062} C_VEL
LIN {X 0,Y 466.777,Z 273.47,A -85,B 0,C 180,E1 -7456.947,E2 -7456.947} C_VEL
LIN {X 0,Y 466.745,Z 275.009,A -85,B 0,C 180,E1 -7458.163,E2 -7458.163} C_VEL
LIN {X 0,Y 466.679,Z 275.818,A -85,B 0,C 180,E1 -7459.589,E2 -7459.589} C_VEL
LIN {X 0,Y 466.712,Z 275.372,A -85,B 0,C 180,E1 -7461.339,E2 -7461.339} C_VEL
LIN {X 0,Y 466.753,Z 274.518,A -85,B 0,C 180,E1 -7462.212,E2 -7462.212} C_VEL
LIN {X 0,Y 466.871,Z 272.582,A -85,B 0,C 180,E1 -7463.476,E2 -7463.476} C_VEL
LIN {X 0,Y 466.881,Z 269.532,A -85,B 0,C 180,E1 -7464.818,E2 -7464.818} C_VEL
LIN {X 0,Y 467.113,Z 265.511,A -85,B 0,C 180,E1 -7466.118,E2 -7466.118} C_VEL
LIN {X 0,Y 467.201,Z 260.367,A -85,B 0,C 180,E1 -7467.414,E2 -7467.414} C_VEL
LIN {X 0,Y 467.544,Z 253.889,A -85,B 0,C 180,E1 -7468.708,E2 -7468.708} C_VEL
LIN {X 0,Y 467.918,Z 245.862,A -85,B 0,C 180,E1 -7470,E2 -7470} C_VEL
LIN {X 0,Y 468.257,Z 237.685,A -85,B 0,C 180,E1 -7471.075,E2 -7471.075} C_VEL
LIN {X 0,Y 468.788,Z 227.654,A -85,B 0,C 180,E1 -7472.148,E2 -7472.148} C_VEL
LIN {X 0,Y 469.274,Z 217.722,A -85,B 0,C 180,E1 -7473.005,E2 -7473.005} C_VEL
LIN {X 0,Y 469.737,Z 206.935,A -85,B 0,C 180,E1 -7473.753,E2 -7473.753} C_VEL
